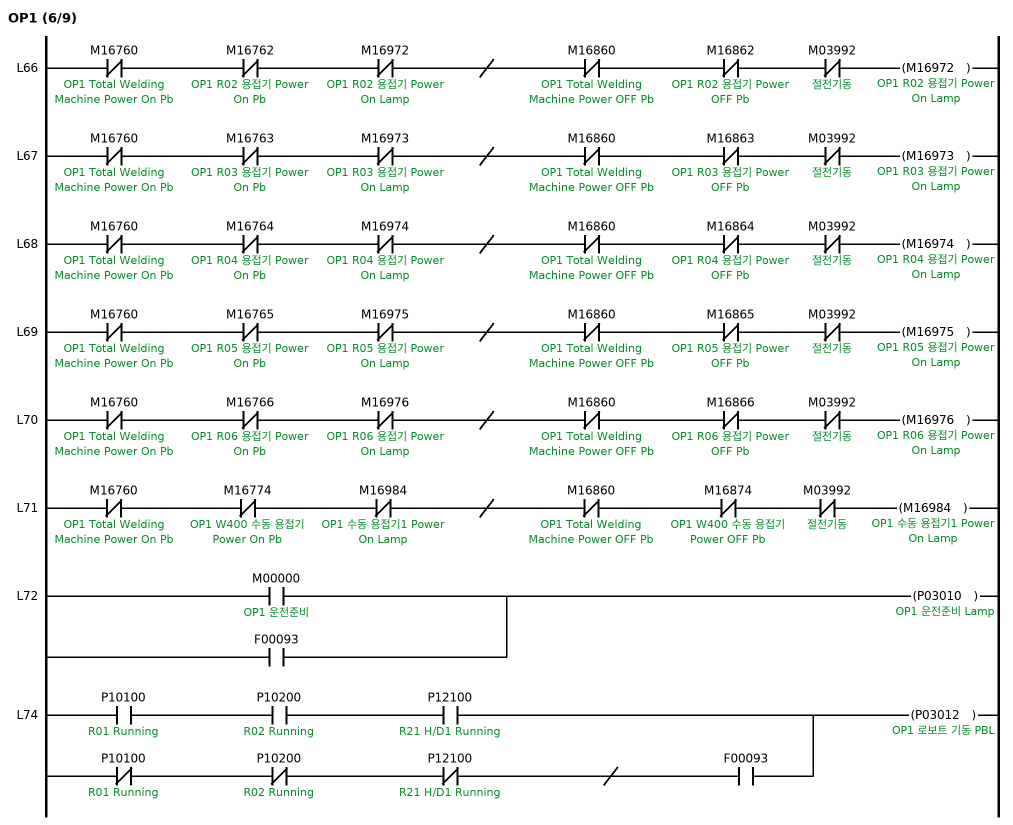
; L66
LOAD NOT  M16760	// OP1 Total Welding Machine Power On Pb
AND NOT   M16762	// OP1 R02 용접기 Power On Pb
AND NOT   M16972	// OP1 R02 용접기 Power On Lamp
NOT
AND NOT   M16860	// OP1 Total Welding Machine Power OFF Pb
AND NOT   M16862	// OP1 R02 용접기 Power OFF Pb
AND NOT   M03992	// 절전기동
OUT       M16972	// OP1 R02 용접기 Power On Lamp
; L67
LOAD NOT  M16760	// OP1 Total Welding Machine Power On Pb
AND NOT   M16763	// OP1 R03 용접기 Power On Pb
AND NOT   M16973	// OP1 R03 용접기 Power On Lamp
NOT
AND NOT   M16860	// OP1 Total Welding Machine Power OFF Pb
AND NOT   M16863	// OP1 R03 용접기 Power OFF Pb
AND NOT   M03992	// 절전기동
OUT       M16973	// OP1 R03 용접기 Power On Lamp
; L68
LOAD NOT  M16760	// OP1 Total Welding Machine Power On Pb
AND NOT   M16764	// OP1 R04 용접기 Power On Pb
AND NOT   M16974	// OP1 R04 용접기 Power On Lamp
NOT
AND NOT   M16860	// OP1 Total Welding Machine Power OFF Pb
AND NOT   M16864	// OP1 R04 용접기 Power OFF Pb
AND NOT   M03992	// 절전기동
OUT       M16974	// OP1 R04 용접기 Power On Lamp
; L69
LOAD NOT  M16760	// OP1 Total Welding Machine Power On Pb
AND NOT   M16765	// OP1 R05 용접기 Power On Pb
AND NOT   M16975	// OP1 R05 용접기 Power On Lamp
NOT
AND NOT   M16860	// OP1 Total Welding Machine Power OFF Pb
AND NOT   M16865	// OP1 R05 용접기 Power OFF Pb
AND NOT   M03992	// 절전기동
OUT       M16975	// OP1 R05 용접기 Power On Lamp
; L70
LOAD NOT  M16760	// OP1 Total Welding Machine Power On Pb
AND NOT   M16766	// OP1 R06 용접기 Power On Pb
AND NOT   M16976	// OP1 R06 용접기 Power On Lamp
NOT
AND NOT   M16860	// OP1 Total Welding Machine Power OFF Pb
AND NOT   M16866	// OP1 R06 용접기 Power OFF Pb
AND NOT   M03992	// 절전기동
OUT       M16976	// OP1 R06 용접기 Power On Lamp
; L71
LOAD NOT  M16760	// OP1 Total Welding Machine Power On Pb
AND NOT   M16774	// OP1 W400 수동 용접기 Power On Pb
AND NOT   M16984	// OP1 수동 용접기1 Power On Lamp
NOT
AND NOT   M16860	// OP1 Total Welding Machine Power OFF Pb
AND NOT   M16874	// OP1 W400 수동 용접기 Power OFF Pb
AND NOT   M03992	// 절전기동
OUT       M16984	// OP1 수동 용접기1 Power On Lamp
; L72
LOAD      M00000	// OP1 운전준비
OR        F00093
OUT       P03010	// OP1 운전준비 Lamp
; L74
LOAD      P10100	// R01 Running
AND       P10200	// R02 Running
AND       P12100	// R21 H/D1 Running
LOAD NOT  P10100	// R01 Running
AND NOT   P10200	// R02 Running
AND NOT   P12100	// R21 H/D1 Running
NOT
AND       F00093
OR LOAD
OUT       P03012	// OP1 로보트 기동 PBL

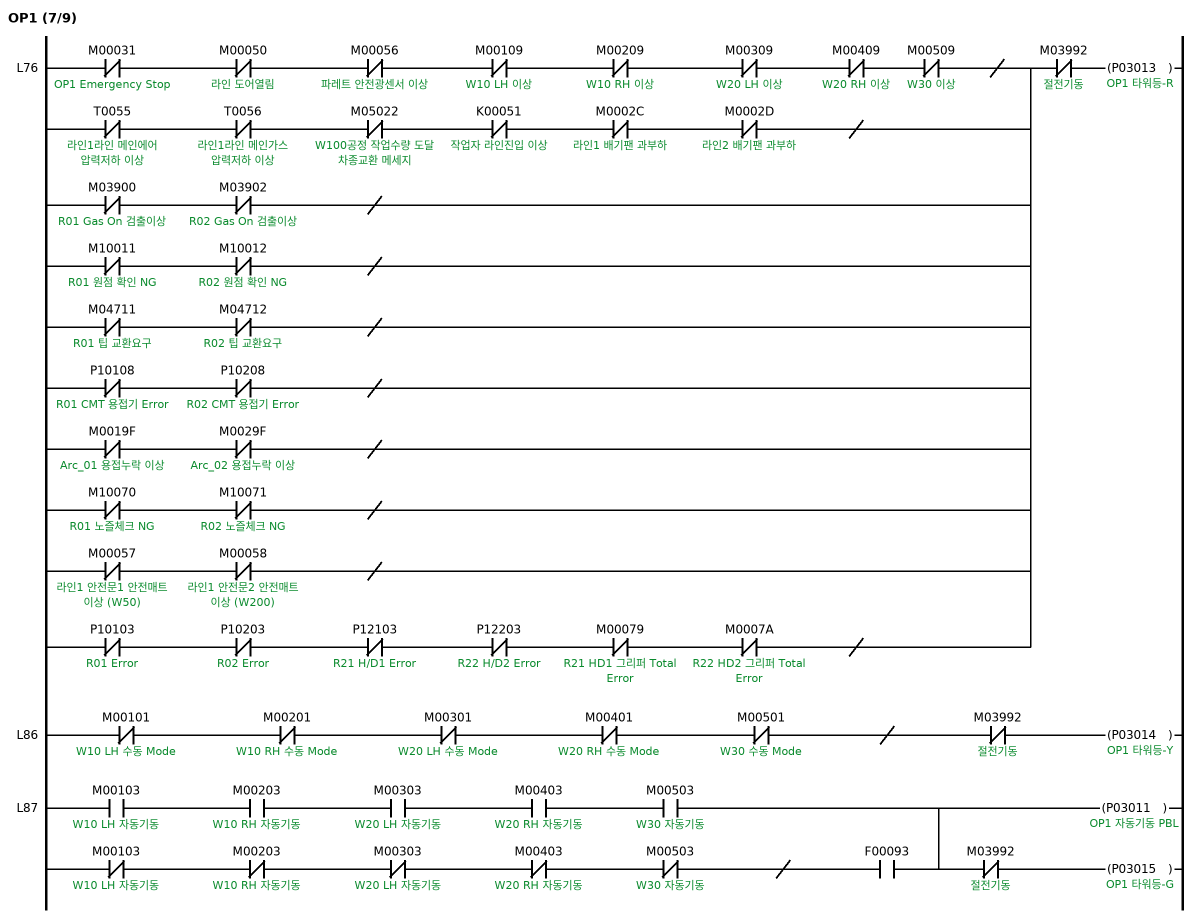
; L76
LOAD NOT  M00031	// OP1 Emergency Stop
AND NOT   M00050	// 라인 도어열림
AND NOT   M00056	// 파레트 안전광센서 이상
AND NOT   M00109	// W10 LH 이상
AND NOT   M00209	// W10 RH 이상
AND NOT   M00309	// W20 LH 이상
AND NOT   M00409	// W20 RH 이상
AND NOT   M00509	// W30 이상
NOT
LOAD NOT  T0055	// 라인1라인 메인에어 압력저하 이상
AND NOT   T0056	// 라인1라인 메인가스 압력저하 이상
AND NOT   M05022	// W100공정 작업수량 도달 차종교환 메세지
AND NOT   K00051	//  작업자 라인진입 이상
AND NOT   M0002C	// 라인1 배기팬 과부하
AND NOT   M0002D	// 라인2 배기팬 과부하
NOT
OR LOAD
LOAD NOT  M03900	// R01 Gas On 검출이상
AND NOT   M03902	// R02 Gas On 검출이상
NOT
OR LOAD
LOAD NOT  M10011	// R01 원점 확인 NG
AND NOT   M10012	// R02 원점 확인 NG
NOT
OR LOAD
LOAD NOT  M04711	// R01 팁 교환요구
AND NOT   M04712	// R02 팁 교환요구
NOT
OR LOAD
LOAD NOT  P10108	// R01 CMT 용접기 Error
AND NOT   P10208	// R02 CMT 용접기 Error
NOT
OR LOAD
LOAD NOT  M0019F	// Arc_01 용접누락 이상
AND NOT   M0029F	// Arc_02 용접누락 이상
NOT
OR LOAD
LOAD NOT  M10070	// R01 노즐체크 NG
AND NOT   M10071	// R02 노즐체크 NG
NOT
OR LOAD
LOAD NOT  M00057	// 라인1 안전문1 안전매트 이상 (W50)
AND NOT   M00058	// 라인1 안전문2 안전매트 이상 (W200)
NOT
OR LOAD
LOAD NOT  P10103	// R01 Error
AND NOT   P10203	// R02 Error
AND NOT   P12103	// R21 H/D1 Error
AND NOT   P12203	// R22 H/D2 Error
AND NOT   M00079	// R21 HD1 그리퍼 Total Error 
AND NOT   M0007A	// R22 HD2 그리퍼 Total Error 
NOT
OR LOAD
AND NOT   M03992	// 절전기동
OUT       P03013	// OP1 타워등-R
; L86
LOAD NOT  M00101	// W10 LH 수동 Mode
AND NOT   M00201	// W10 RH 수동 Mode
AND NOT   M00301	// W20 LH 수동 Mode
AND NOT   M00401	// W20 RH 수동 Mode
AND NOT   M00501	// W30 수동 Mode
NOT
AND NOT   M03992	// 절전기동
OUT       P03014	// OP1 타워등-Y
; L87
LOAD      M00103	// W10 LH 자동기동
AND       M00203	// W10 RH 자동기동
AND       M00303	// W20 LH 자동기동
AND       M00403	// W20 RH 자동기동
AND       M00503	// W30 자동기동
LOAD NOT  M00103	// W10 LH 자동기동
AND NOT   M00203	// W10 RH 자동기동
AND NOT   M00303	// W20 LH 자동기동
AND NOT   M00403	// W20 RH 자동기동
AND NOT   M00503	// W30 자동기동
NOT
AND       F00093
OR LOAD
OUT       P03011	// OP1 자동기동 PBL
AND NOT   M03992	// 절전기동
OUT       P03015	// OP1 타워등-G

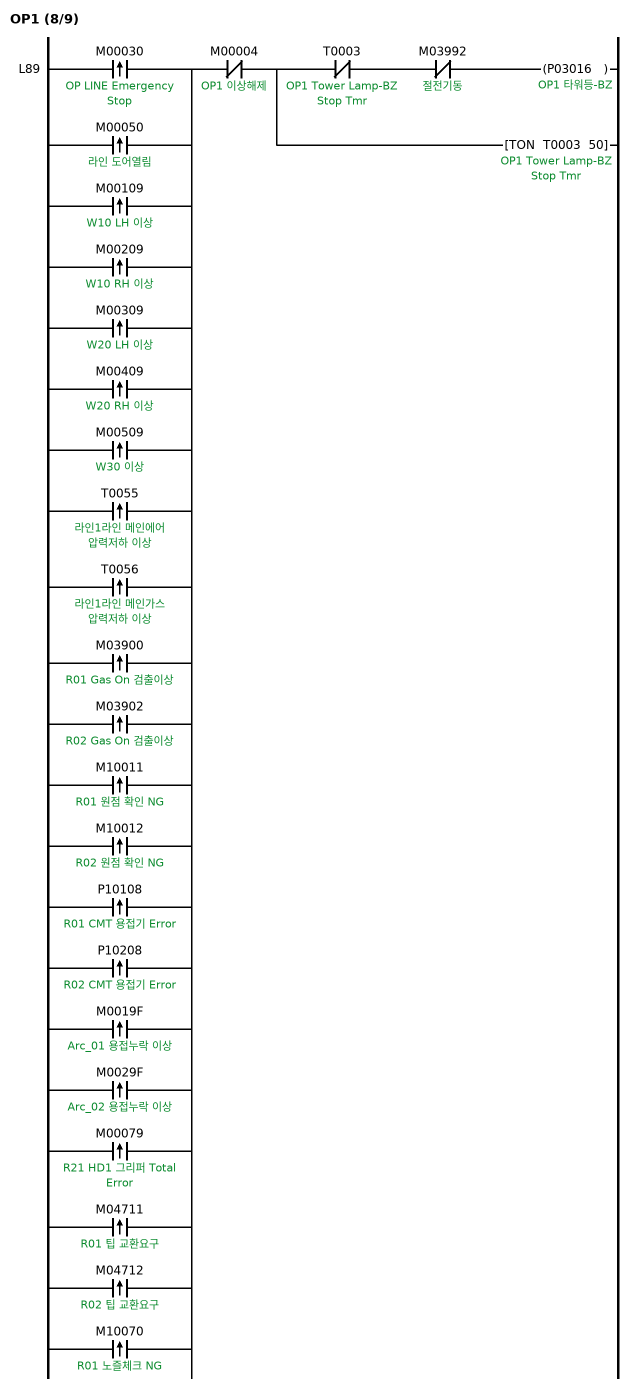

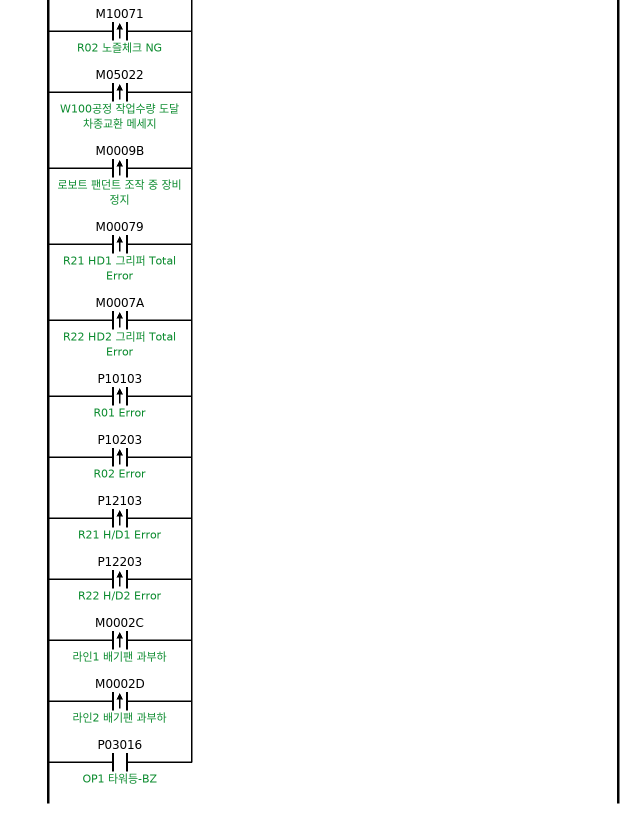
; L89
LOADP     M00030	// OP LINE Emergency Stop
ORP       M00050	// 라인 도어열림
ORP       M00109	// W10 LH 이상
ORP       M00209	// W10 RH 이상
ORP       M00309	// W20 LH 이상
ORP       M00409	// W20 RH 이상
ORP       M00509	// W30 이상
ORP       T0055	// 라인1라인 메인에어 압력저하 이상
ORP       T0056	// 라인1라인 메인가스 압력저하 이상
ORP       M03900	// R01 Gas On 검출이상
ORP       M03902	// R02 Gas On 검출이상
ORP       M10011	// R01 원점 확인 NG
ORP       M10012	// R02 원점 확인 NG
ORP       P10108	// R01 CMT 용접기 Error
ORP       P10208	// R02 CMT 용접기 Error
ORP       M0019F	// Arc_01 용접누락 이상
ORP       M0029F	// Arc_02 용접누락 이상
ORP       M00079	// R21 HD1 그리퍼 Total Error 
ORP       M04711	// R01 팁 교환요구
ORP       M04712	// R02 팁 교환요구
ORP       M10070	// R01 노즐체크 NG
ORP       M10071	// R02 노즐체크 NG
ORP       M05022	// W100공정 작업수량 도달 차종교환 메세지
ORP       M0009B	// 로보트 팬던트 조작 중 장비 정지
ORP       M00079	// R21 HD1 그리퍼 Total Error 
ORP       M0007A	// R22 HD2 그리퍼 Total Error 
ORP       P10103	// R01 Error
ORP       P10203	// R02 Error
ORP       P12103	// R21 H/D1 Error
ORP       P12203	// R22 H/D2 Error
ORP       M0002C	// 라인1 배기팬 과부하
ORP       M0002D	// 라인2 배기팬 과부하
OR        P03016	// OP1 타워등-BZ
AND NOT   M00004	// OP1 이상해제
MPUSH
AND NOT   T0003	// OP1 Tower Lamp-BZ Stop Tmr
AND NOT   M03992	// 절전기동
OUT       P03016	// OP1 타워등-BZ
MPOP
TON       T0003 50	// OP1 Tower Lamp-BZ Stop Tmr

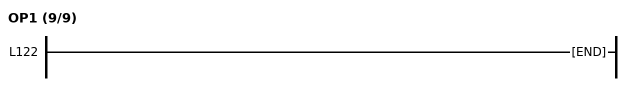
; L122
END

PROGRAM OP2 (task: 스캔 프로그램)

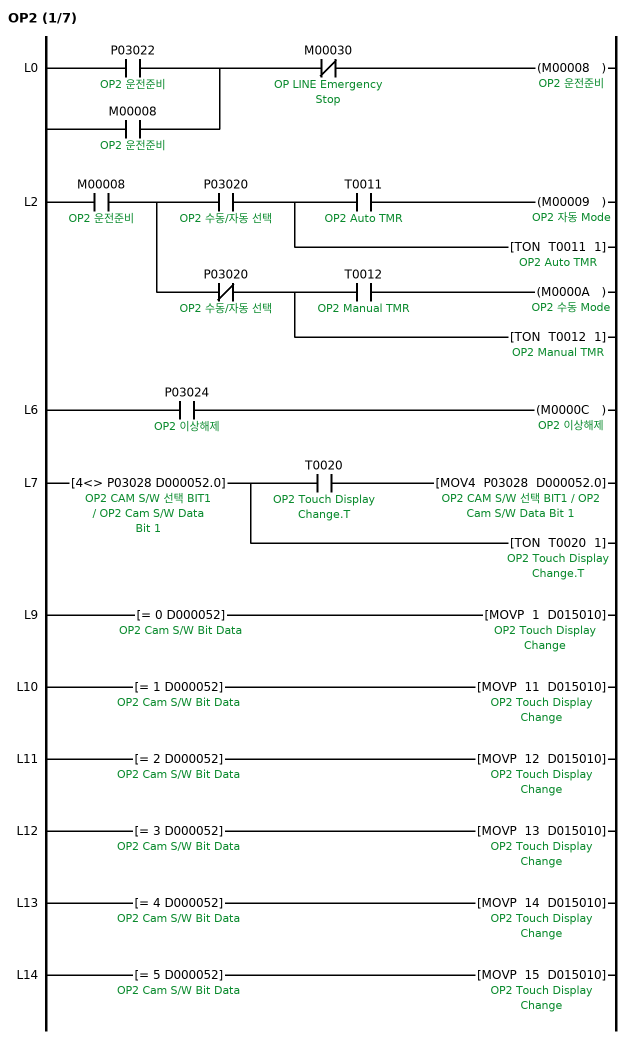
; L0
LOAD      P03022	// OP2 운전준비
OR        M00008	// OP2 운전준비
AND NOT   M00030	// OP LINE Emergency Stop
OUT       M00008	// OP2 운전준비
; L2
LOAD      M00008	// OP2 운전준비
MPUSH
AND       P03020	// OP2 수동/자동 선택
MPUSH
AND       T0011	// OP2 Auto TMR
OUT       M00009	// OP2 자동 Mode
MPOP
TON       T0011 1	// OP2 Auto TMR
MPOP
AND NOT   P03020	// OP2 수동/자동 선택
MPUSH
AND       T0012	// OP2 Manual TMR
OUT       M0000A	// OP2 수동 Mode
MPOP
TON       T0012 1	// OP2 Manual TMR
; L6
LOAD      P03024	// OP2 이상해제
OUT       M0000C	// OP2 이상해제
; L7
LOAD4<>   P03028 D000052.0	// OP2 CAM S/W 선택 BIT1 / OP2 Cam S/W Data Bit 1
MPUSH
AND       T0020	// OP2 Touch Display Change.T
MOV4      P03028 D000052.0	// OP2 CAM S/W 선택 BIT1 / OP2 Cam S/W Data Bit 1
MPOP
TON       T0020 1	// OP2 Touch Display Change.T
; L9
LOAD=     0 D000052	// OP2 Cam S/W Bit Data
MOVP      1 D015010	// OP2 Touch Display Change
; L10
LOAD=     1 D000052	// OP2 Cam S/W Bit Data
MOVP      11 D015010	// OP2 Touch Display Change
; L11
LOAD=     2 D000052	// OP2 Cam S/W Bit Data
MOVP      12 D015010	// OP2 Touch Display Change
; L12
LOAD=     3 D000052	// OP2 Cam S/W Bit Data
MOVP      13 D015010	// OP2 Touch Display Change
; L13
LOAD=     4 D000052	// OP2 Cam S/W Bit Data
MOVP      14 D015010	// OP2 Touch Display Change
; L14
LOAD=     5 D000052	// OP2 Cam S/W Bit Data
MOVP      15 D015010	// OP2 Touch Display Change

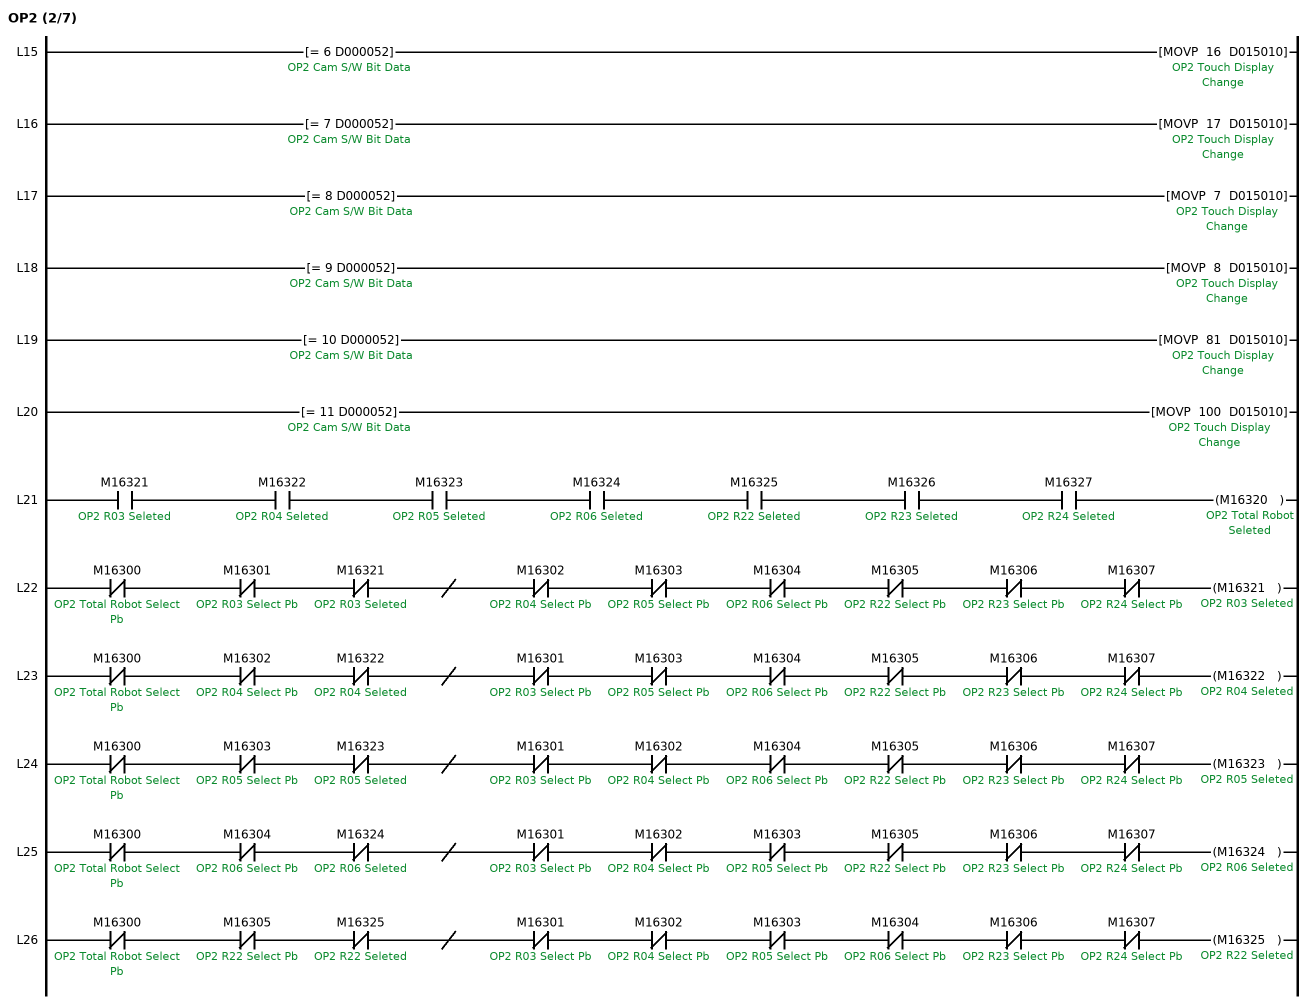
; L15
LOAD=     6 D000052	// OP2 Cam S/W Bit Data
MOVP      16 D015010	// OP2 Touch Display Change
; L16
LOAD=     7 D000052	// OP2 Cam S/W Bit Data
MOVP      17 D015010	// OP2 Touch Display Change
; L17
LOAD=     8 D000052	// OP2 Cam S/W Bit Data
MOVP      7 D015010	// OP2 Touch Display Change
; L18
LOAD=     9 D000052	// OP2 Cam S/W Bit Data
MOVP      8 D015010	// OP2 Touch Display Change
; L19
LOAD=     10 D000052	// OP2 Cam S/W Bit Data
MOVP      81 D015010	// OP2 Touch Display Change
; L20
LOAD=     11 D000052	// OP2 Cam S/W Bit Data
MOVP      100 D015010	// OP2 Touch Display Change
; L21
LOAD      M16321	// OP2 R03 Seleted
AND       M16322	// OP2 R04 Seleted
AND       M16323	// OP2 R05 Seleted
AND       M16324	// OP2 R06 Seleted
AND       M16325	// OP2 R22 Seleted
AND       M16326	// OP2 R23 Seleted
AND       M16327	// OP2 R24 Seleted
OUT       M16320	// OP2 Total Robot Seleted
; L22
LOAD NOT  M16300	// OP2 Total Robot Select Pb
AND NOT   M16301	// OP2 R03 Select Pb
AND NOT   M16321	// OP2 R03 Seleted
NOT
AND NOT   M16302	// OP2 R04 Select Pb
AND NOT   M16303	// OP2 R05 Select Pb
AND NOT   M16304	// OP2 R06 Select Pb
AND NOT   M16305	// OP2 R22 Select Pb
AND NOT   M16306	// OP2 R23 Select Pb
AND NOT   M16307	// OP2 R24 Select Pb
OUT       M16321	// OP2 R03 Seleted
; L23
LOAD NOT  M16300	// OP2 Total Robot Select Pb
AND NOT   M16302	// OP2 R04 Select Pb
AND NOT   M16322	// OP2 R04 Seleted
NOT
AND NOT   M16301	// OP2 R03 Select Pb
AND NOT   M16303	// OP2 R05 Select Pb
AND NOT   M16304	// OP2 R06 Select Pb
AND NOT   M16305	// OP2 R22 Select Pb
AND NOT   M16306	// OP2 R23 Select Pb
AND NOT   M16307	// OP2 R24 Select Pb
OUT       M16322	// OP2 R04 Seleted
; L24
LOAD NOT  M16300	// OP2 Total Robot Select Pb
AND NOT   M16303	// OP2 R05 Select Pb
AND NOT   M16323	// OP2 R05 Seleted
NOT
AND NOT   M16301	// OP2 R03 Select Pb
AND NOT   M16302	// OP2 R04 Select Pb
AND NOT   M16304	// OP2 R06 Select Pb
AND NOT   M16305	// OP2 R22 Select Pb
AND NOT   M16306	// OP2 R23 Select Pb
AND NOT   M16307	// OP2 R24 Select Pb
OUT       M16323	// OP2 R05 Seleted
; L25
LOAD NOT  M16300	// OP2 Total Robot Select Pb
AND NOT   M16304	// OP2 R06 Select Pb
AND NOT   M16324	// OP2 R06 Seleted
NOT
AND NOT   M16301	// OP2 R03 Select Pb
AND NOT   M16302	// OP2 R04 Select Pb
AND NOT   M16303	// OP2 R05 Select Pb
AND NOT   M16305	// OP2 R22 Select Pb
AND NOT   M16306	// OP2 R23 Select Pb
AND NOT   M16307	// OP2 R24 Select Pb
OUT       M16324	// OP2 R06 Seleted
; L26
LOAD NOT  M16300	// OP2 Total Robot Select Pb
AND NOT   M16305	// OP2 R22 Select Pb
AND NOT   M16325	// OP2 R22 Seleted
NOT
AND NOT   M16301	// OP2 R03 Select Pb
AND NOT   M16302	// OP2 R04 Select Pb
AND NOT   M16303	// OP2 R05 Select Pb
AND NOT   M16304	// OP2 R06 Select Pb
AND NOT   M16306	// OP2 R23 Select Pb
AND NOT   M16307	// OP2 R24 Select Pb
OUT       M16325	// OP2 R22 Seleted

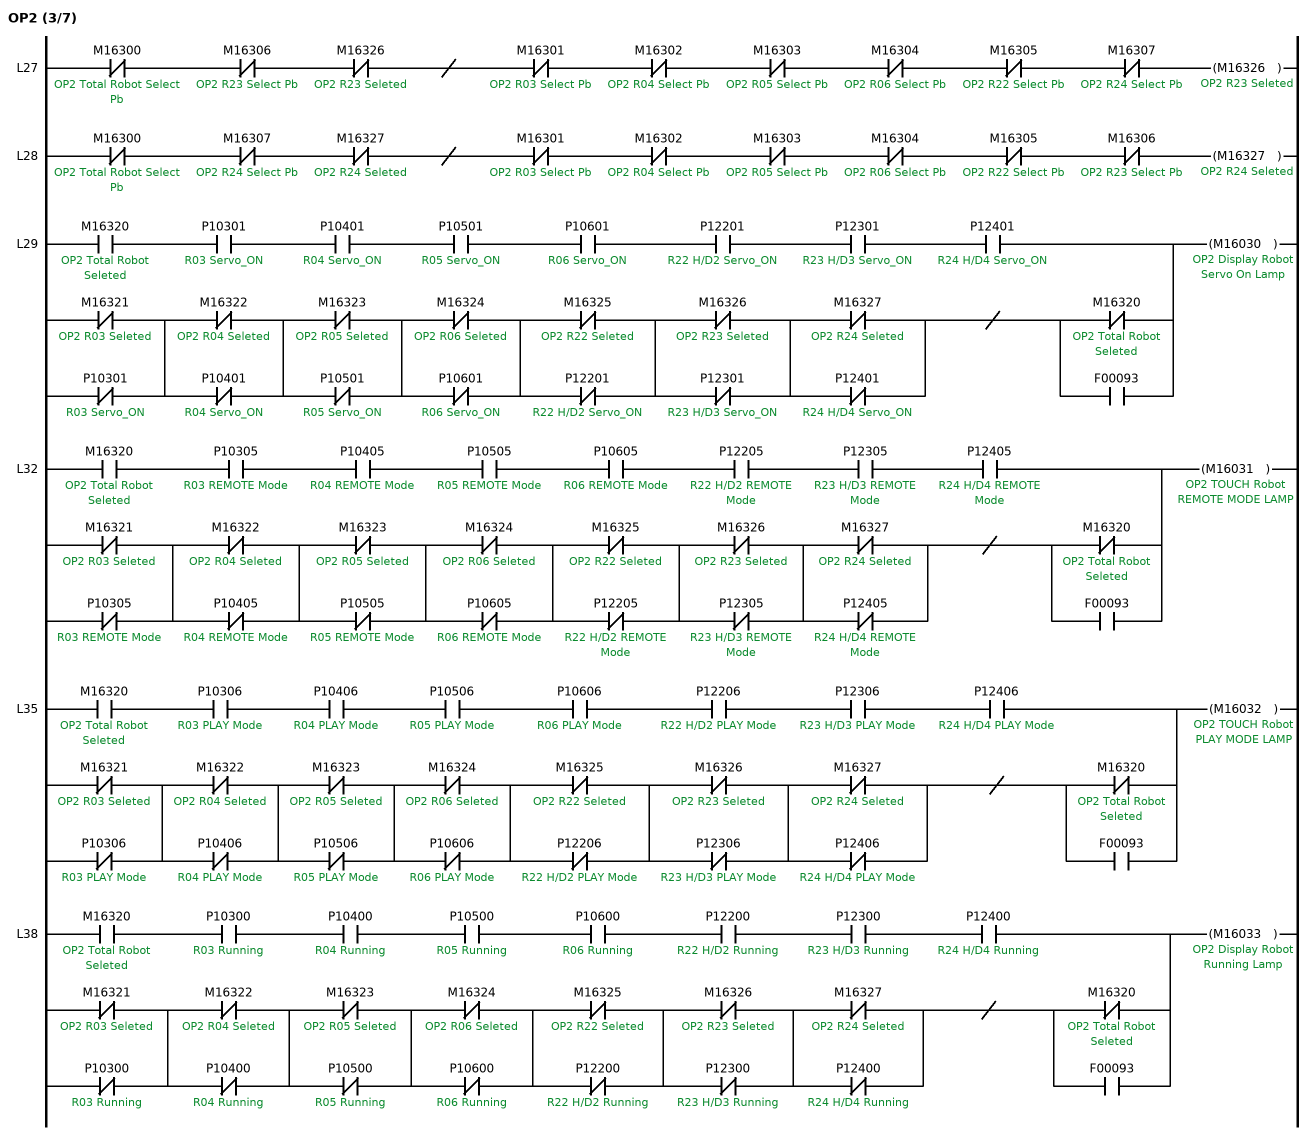
; L27
LOAD NOT  M16300	// OP2 Total Robot Select Pb
AND NOT   M16306	// OP2 R23 Select Pb
AND NOT   M16326	// OP2 R23 Seleted
NOT
AND NOT   M16301	// OP2 R03 Select Pb
AND NOT   M16302	// OP2 R04 Select Pb
AND NOT   M16303	// OP2 R05 Select Pb
AND NOT   M16304	// OP2 R06 Select Pb
AND NOT   M16305	// OP2 R22 Select Pb
AND NOT   M16307	// OP2 R24 Select Pb
OUT       M16326	// OP2 R23 Seleted
; L28
LOAD NOT  M16300	// OP2 Total Robot Select Pb
AND NOT   M16307	// OP2 R24 Select Pb
AND NOT   M16327	// OP2 R24 Seleted
NOT
AND NOT   M16301	// OP2 R03 Select Pb
AND NOT   M16302	// OP2 R04 Select Pb
AND NOT   M16303	// OP2 R05 Select Pb
AND NOT   M16304	// OP2 R06 Select Pb
AND NOT   M16305	// OP2 R22 Select Pb
AND NOT   M16306	// OP2 R23 Select Pb
OUT       M16327	// OP2 R24 Seleted
; L29
LOAD      M16320	// OP2 Total Robot Seleted
AND       P10301	// R03 Servo_ON
AND       P10401	// R04 Servo_ON
AND       P10501	// R05 Servo_ON
AND       P10601	// R06 Servo_ON
AND       P12201	// R22 H/D2 Servo_ON
AND       P12301	// R23 H/D3 Servo_ON
AND       P12401	// R24 H/D4 Servo_ON
LOAD NOT  M16321	// OP2 R03 Seleted
OR NOT    P10301	// R03 Servo_ON
LOAD NOT  M16322	// OP2 R04 Seleted
OR NOT    P10401	// R04 Servo_ON
AND LOAD
LOAD NOT  M16323	// OP2 R05 Seleted
OR NOT    P10501	// R05 Servo_ON
AND LOAD
LOAD NOT  M16324	// OP2 R06 Seleted
OR NOT    P10601	// R06 Servo_ON
AND LOAD
LOAD NOT  M16325	// OP2 R22 Seleted
OR NOT    P12201	// R22 H/D2 Servo_ON
AND LOAD
LOAD NOT  M16326	// OP2 R23 Seleted
OR NOT    P12301	// R23 H/D3 Servo_ON
AND LOAD
LOAD NOT  M16327	// OP2 R24 Seleted
OR NOT    P12401	// R24 H/D4 Servo_ON
AND LOAD
NOT
LOAD NOT  M16320	// OP2 Total Robot Seleted
OR        F00093
AND LOAD
OR LOAD
OUT       M16030	// OP2 Display Robot Servo On Lamp
; L32
LOAD      M16320	// OP2 Total Robot Seleted
AND       P10305	// R03 REMOTE Mode
AND       P10405	// R04 REMOTE Mode
AND       P10505	// R05 REMOTE Mode
AND       P10605	// R06 REMOTE Mode
AND       P12205	// R22 H/D2 REMOTE Mode
AND       P12305	// R23 H/D3 REMOTE Mode
AND       P12405	// R24 H/D4 REMOTE Mode
LOAD NOT  M16321	// OP2 R03 Seleted
OR NOT    P10305	// R03 REMOTE Mode
LOAD NOT  M16322	// OP2 R04 Seleted
OR NOT    P10405	// R04 REMOTE Mode
AND LOAD
LOAD NOT  M16323	// OP2 R05 Seleted
OR NOT    P10505	// R05 REMOTE Mode
AND LOAD
LOAD NOT  M16324	// OP2 R06 Seleted
OR NOT    P10605	// R06 REMOTE Mode
AND LOAD
LOAD NOT  M16325	// OP2 R22 Seleted
OR NOT    P12205	// R22 H/D2 REMOTE Mode
AND LOAD
LOAD NOT  M16326	// OP2 R23 Seleted
OR NOT    P12305	// R23 H/D3 REMOTE Mode
AND LOAD
LOAD NOT  M16327	// OP2 R24 Seleted
OR NOT    P12405	// R24 H/D4 REMOTE Mode
AND LOAD
NOT
LOAD NOT  M16320	// OP2 Total Robot Seleted
OR        F00093
AND LOAD
OR LOAD
OUT       M16031	// OP2 TOUCH Robot REMOTE MODE LAMP
; L35
LOAD      M16320	// OP2 Total Robot Seleted
AND       P10306	// R03 PLAY Mode
AND       P10406	// R04 PLAY Mode
AND       P10506	// R05 PLAY Mode
AND       P10606	// R06 PLAY Mode
AND       P12206	// R22 H/D2 PLAY Mode
AND       P12306	// R23 H/D3 PLAY Mode
AND       P12406	// R24 H/D4 PLAY Mode
LOAD NOT  M16321	// OP2 R03 Seleted
OR NOT    P10306	// R03 PLAY Mode
LOAD NOT  M16322	// OP2 R04 Seleted
OR NOT    P10406	// R04 PLAY Mode
AND LOAD
LOAD NOT  M16323	// OP2 R05 Seleted
OR NOT    P10506	// R05 PLAY Mode
AND LOAD
LOAD NOT  M16324	// OP2 R06 Seleted
OR NOT    P10606	// R06 PLAY Mode
AND LOAD
LOAD NOT  M16325	// OP2 R22 Seleted
OR NOT    P12206	// R22 H/D2 PLAY Mode
AND LOAD
LOAD NOT  M16326	// OP2 R23 Seleted
OR NOT    P12306	// R23 H/D3 PLAY Mode
AND LOAD
LOAD NOT  M16327	// OP2 R24 Seleted
OR NOT    P12406	// R24 H/D4 PLAY Mode
AND LOAD
NOT
LOAD NOT  M16320	// OP2 Total Robot Seleted
OR        F00093
AND LOAD
OR LOAD
OUT       M16032	// OP2 TOUCH Robot PLAY MODE LAMP
; L38
LOAD      M16320	// OP2 Total Robot Seleted
AND       P10300	// R03 Running
AND       P10400	// R04 Running
AND       P10500	// R05 Running
AND       P10600	// R06 Running
AND       P12200	// R22 H/D2 Running
AND       P12300	// R23 H/D3 Running
AND       P12400	// R24 H/D4 Running
LOAD NOT  M16321	// OP2 R03 Seleted
OR NOT    P10300	// R03 Running
LOAD NOT  M16322	// OP2 R04 Seleted
OR NOT    P10400	// R04 Running
AND LOAD
LOAD NOT  M16323	// OP2 R05 Seleted
OR NOT    P10500	// R05 Running
AND LOAD
LOAD NOT  M16324	// OP2 R06 Seleted
OR NOT    P10600	// R06 Running
AND LOAD
LOAD NOT  M16325	// OP2 R22 Seleted
OR NOT    P12200	// R22 H/D2 Running
AND LOAD
LOAD NOT  M16326	// OP2 R23 Seleted
OR NOT    P12300	// R23 H/D3 Running
AND LOAD
LOAD NOT  M16327	// OP2 R24 Seleted
OR NOT    P12400	// R24 H/D4 Running
AND LOAD
NOT
LOAD NOT  M16320	// OP2 Total Robot Seleted
OR        F00093
AND LOAD
OR LOAD
OUT       M16033	// OP2 Display Robot Running Lamp

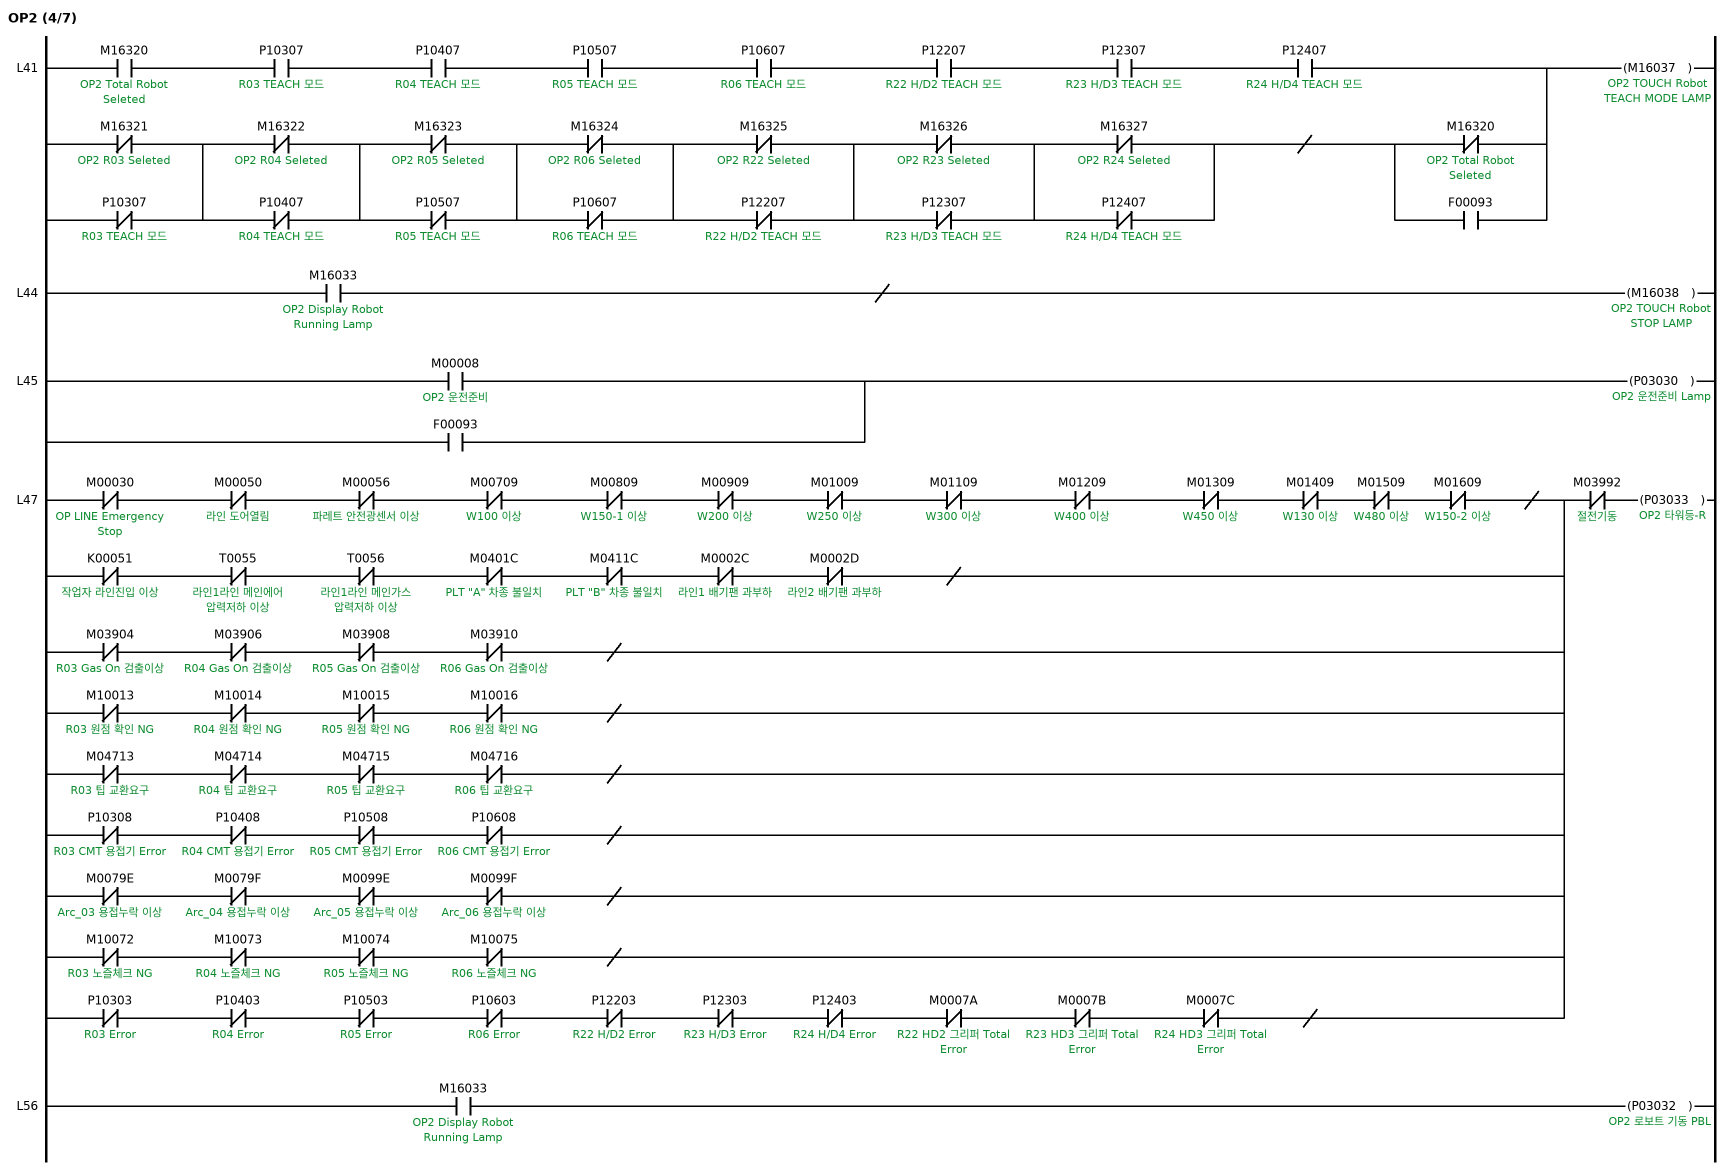
; L41
LOAD      M16320	// OP2 Total Robot Seleted
AND       P10307	// R03 TEACH 모드
AND       P10407	// R04 TEACH 모드
AND       P10507	// R05 TEACH 모드
AND       P10607	// R06 TEACH 모드
AND       P12207	// R22 H/D2 TEACH 모드
AND       P12307	// R23 H/D3 TEACH 모드
AND       P12407	// R24 H/D4 TEACH 모드
LOAD NOT  M16321	// OP2 R03 Seleted
OR NOT    P10307	// R03 TEACH 모드
LOAD NOT  M16322	// OP2 R04 Seleted
OR NOT    P10407	// R04 TEACH 모드
AND LOAD
LOAD NOT  M16323	// OP2 R05 Seleted
OR NOT    P10507	// R05 TEACH 모드
AND LOAD
LOAD NOT  M16324	// OP2 R06 Seleted
OR NOT    P10607	// R06 TEACH 모드
AND LOAD
LOAD NOT  M16325	// OP2 R22 Seleted
OR NOT    P12207	// R22 H/D2 TEACH 모드
AND LOAD
LOAD NOT  M16326	// OP2 R23 Seleted
OR NOT    P12307	// R23 H/D3 TEACH 모드
AND LOAD
LOAD NOT  M16327	// OP2 R24 Seleted
OR NOT    P12407	// R24 H/D4 TEACH 모드
AND LOAD
NOT
LOAD NOT  M16320	// OP2 Total Robot Seleted
OR        F00093
AND LOAD
OR LOAD
OUT       M16037	// OP2 TOUCH Robot TEACH MODE LAMP
; L44
LOAD      M16033	// OP2 Display Robot Running Lamp
NOT
OUT       M16038	// OP2 TOUCH Robot STOP LAMP
; L45
LOAD      M00008	// OP2 운전준비
OR        F00093
OUT       P03030	// OP2 운전준비 Lamp
; L47
LOAD NOT  M00030	// OP LINE Emergency Stop
AND NOT   M00050	// 라인 도어열림
AND NOT   M00056	// 파레트 안전광센서 이상
AND NOT   M00709	// W100 이상
AND NOT   M00809	// W150-1 이상
AND NOT   M00909	// W200 이상
AND NOT   M01009	// W250 이상
AND NOT   M01109	// W300 이상
AND NOT   M01209	// W400 이상
AND NOT   M01309	// W450 이상
AND NOT   M01409	// W130 이상
AND NOT   M01509	// W480 이상
AND NOT   M01609	// W150-2 이상
NOT
LOAD NOT  K00051	//  작업자 라인진입 이상
AND NOT   T0055	// 라인1라인 메인에어 압력저하 이상
AND NOT   T0056	// 라인1라인 메인가스 압력저하 이상
AND NOT   M0401C	// PLT "A" 차종 불일치
AND NOT   M0411C	// PLT "B" 차종 불일치
AND NOT   M0002C	// 라인1 배기팬 과부하
AND NOT   M0002D	// 라인2 배기팬 과부하
NOT
OR LOAD
LOAD NOT  M03904	// R03 Gas On 검출이상
AND NOT   M03906	// R04 Gas On 검출이상
AND NOT   M03908	// R05 Gas On 검출이상
AND NOT   M03910	// R06 Gas On 검출이상
NOT
OR LOAD
LOAD NOT  M10013	// R03 원점 확인 NG
AND NOT   M10014	// R04 원점 확인 NG
AND NOT   M10015	// R05 원점 확인 NG
AND NOT   M10016	// R06 원점 확인 NG
NOT
OR LOAD
LOAD NOT  M04713	// R03 팁 교환요구
AND NOT   M04714	// R04 팁 교환요구
AND NOT   M04715	// R05 팁 교환요구
AND NOT   M04716	// R06 팁 교환요구
NOT
OR LOAD
LOAD NOT  P10308	// R03 CMT 용접기 Error
AND NOT   P10408	// R04 CMT 용접기 Error
AND NOT   P10508	// R05 CMT 용접기 Error
AND NOT   P10608	// R06 CMT 용접기 Error
NOT
OR LOAD
LOAD NOT  M0079E	// Arc_03 용접누락 이상
AND NOT   M0079F	// Arc_04 용접누락 이상
AND NOT   M0099E	// Arc_05 용접누락 이상
AND NOT   M0099F	// Arc_06 용접누락 이상
NOT
OR LOAD
LOAD NOT  M10072	// R03 노즐체크 NG
AND NOT   M10073	// R04 노즐체크 NG
AND NOT   M10074	// R05 노즐체크 NG
AND NOT   M10075	// R06 노즐체크 NG
NOT
OR LOAD
LOAD NOT  P10303	// R03 Error
AND NOT   P10403	// R04 Error
AND NOT   P10503	// R05 Error
AND NOT   P10603	// R06 Error
AND NOT   P12203	// R22 H/D2 Error
AND NOT   P12303	// R23 H/D3 Error
AND NOT   P12403	// R24 H/D4 Error
AND NOT   M0007A	// R22 HD2 그리퍼 Total Error 
AND NOT   M0007B	// R23 HD3 그리퍼 Total Error 
AND NOT   M0007C	// R24 HD3 그리퍼 Total Error 
NOT
OR LOAD
AND NOT   M03992	// 절전기동
OUT       P03033	// OP2 타워등-R
; L56
LOAD      M16033	// OP2 Display Robot Running Lamp
OUT       P03032	// OP2 로보트 기동 PBL

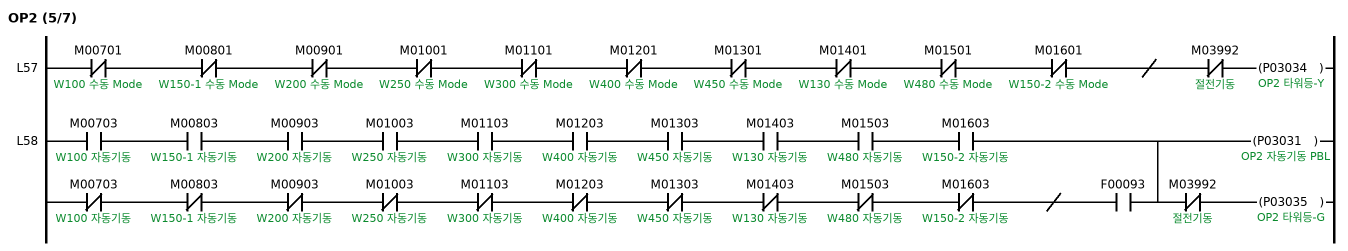
; L57
LOAD NOT  M00701	// W100 수동 Mode
AND NOT   M00801	// W150-1 수동 Mode
AND NOT   M00901	// W200 수동 Mode
AND NOT   M01001	// W250 수동 Mode
AND NOT   M01101	// W300 수동 Mode
AND NOT   M01201	// W400 수동 Mode
AND NOT   M01301	// W450 수동 Mode
AND NOT   M01401	// W130 수동 Mode
AND NOT   M01501	// W480 수동 Mode
AND NOT   M01601	// W150-2 수동 Mode
NOT
AND NOT   M03992	// 절전기동
OUT       P03034	// OP2 타워등-Y
; L58
LOAD      M00703	// W100 자동기동
AND       M00803	// W150-1 자동기동
AND       M00903	// W200 자동기동
AND       M01003	// W250 자동기동
AND       M01103	// W300 자동기동
AND       M01203	// W400 자동기동
AND       M01303	// W450 자동기동
AND       M01403	// W130 자동기동
AND       M01503	// W480 자동기동
AND       M01603	// W150-2 자동기동
LOAD NOT  M00703	// W100 자동기동
AND NOT   M00803	// W150-1 자동기동
AND NOT   M00903	// W200 자동기동
AND NOT   M01003	// W250 자동기동
AND NOT   M01103	// W300 자동기동
AND NOT   M01203	// W400 자동기동
AND NOT   M01303	// W450 자동기동
AND NOT   M01403	// W130 자동기동
AND NOT   M01503	// W480 자동기동
AND NOT   M01603	// W150-2 자동기동
NOT
AND       F00093
OR LOAD
OUT       P03031	// OP2 자동기동 PBL
AND NOT   M03992	// 절전기동
OUT       P03035	// OP2 타워등-G

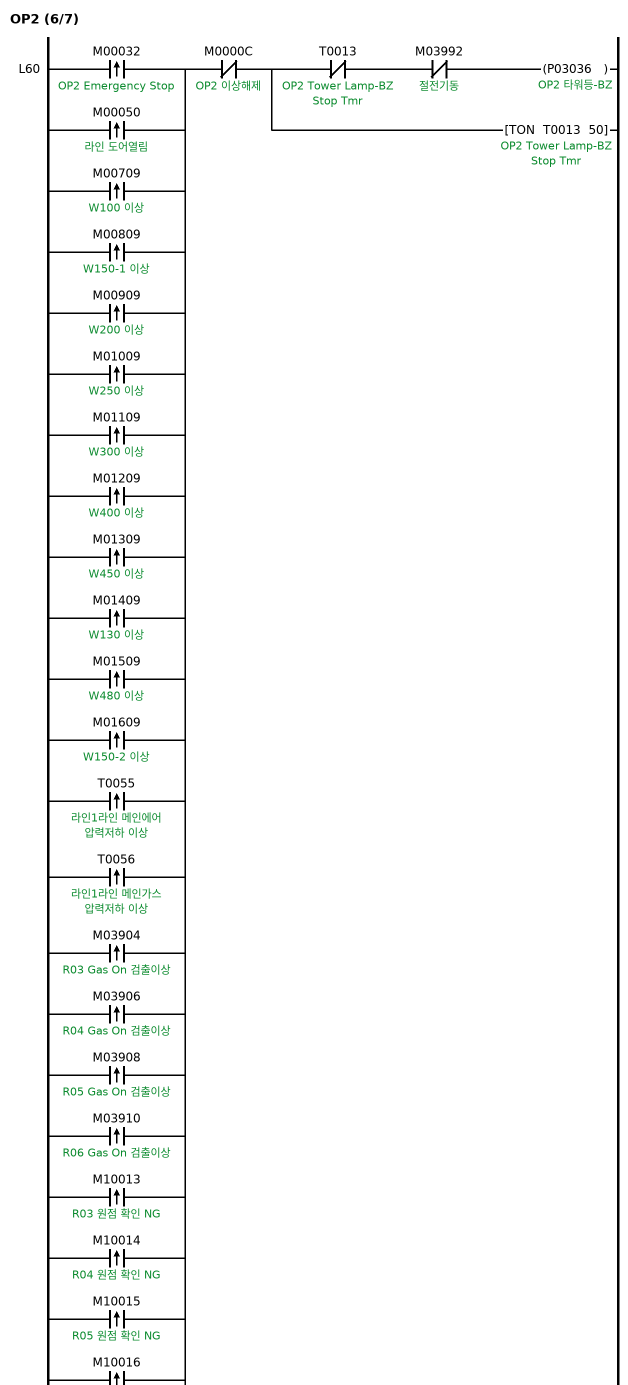

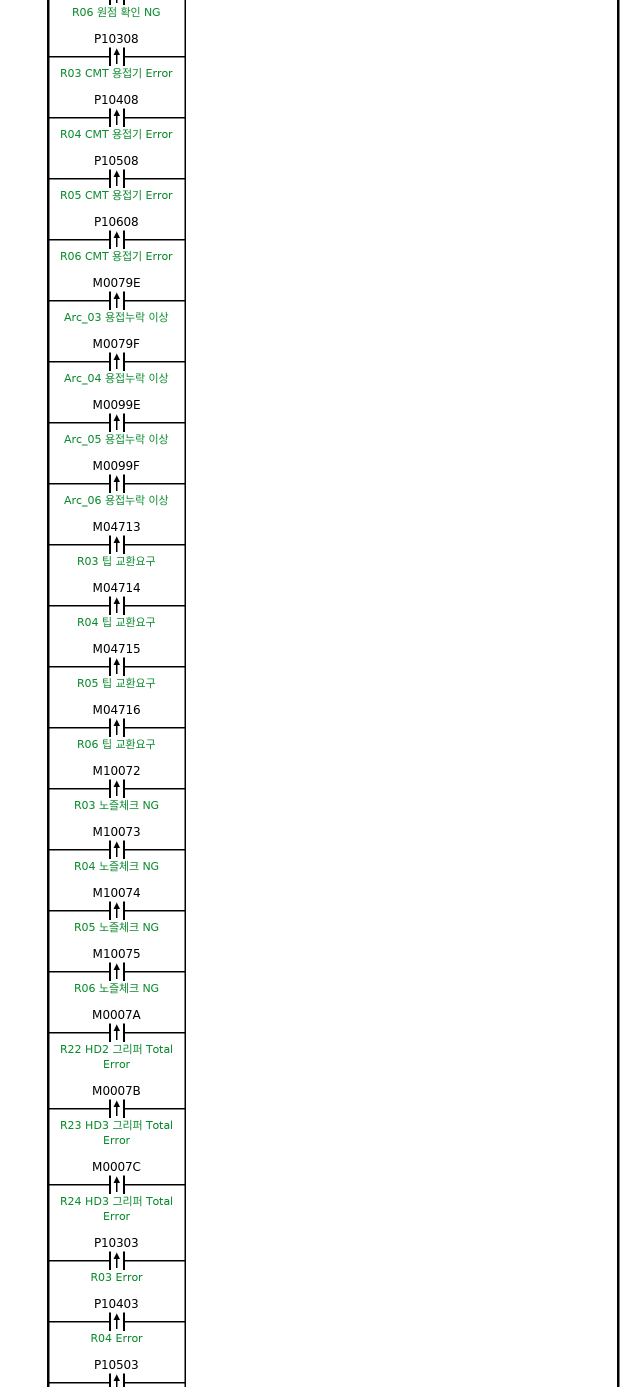

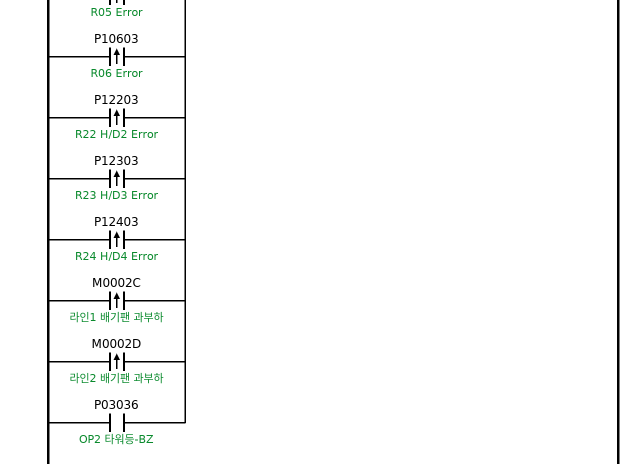
; L60
LOADP     M00032	// OP2 Emergency Stop
ORP       M00050	// 라인 도어열림
ORP       M00709	// W100 이상
ORP       M00809	// W150-1 이상
ORP       M00909	// W200 이상
ORP       M01009	// W250 이상
ORP       M01109	// W300 이상
ORP       M01209	// W400 이상
ORP       M01309	// W450 이상
ORP       M01409	// W130 이상
ORP       M01509	// W480 이상
ORP       M01609	// W150-2 이상
ORP       T0055	// 라인1라인 메인에어 압력저하 이상
ORP       T0056	// 라인1라인 메인가스 압력저하 이상
ORP       M03904	// R03 Gas On 검출이상
ORP       M03906	// R04 Gas On 검출이상
ORP       M03908	// R05 Gas On 검출이상
ORP       M03910	// R06 Gas On 검출이상
ORP       M10013	// R03 원점 확인 NG
ORP       M10014	// R04 원점 확인 NG
ORP       M10015	// R05 원점 확인 NG
ORP       M10016	// R06 원점 확인 NG
ORP       P10308	// R03 CMT 용접기 Error
ORP       P10408	// R04 CMT 용접기 Error
ORP       P10508	// R05 CMT 용접기 Error
ORP       P10608	// R06 CMT 용접기 Error
ORP       M0079E	// Arc_03 용접누락 이상
ORP       M0079F	// Arc_04 용접누락 이상
ORP       M0099E	// Arc_05 용접누락 이상
ORP       M0099F	// Arc_06 용접누락 이상
ORP       M04713	// R03 팁 교환요구
ORP       M04714	// R04 팁 교환요구
ORP       M04715	// R05 팁 교환요구
ORP       M04716	// R06 팁 교환요구
ORP       M10072	// R03 노즐체크 NG
ORP       M10073	// R04 노즐체크 NG
ORP       M10074	// R05 노즐체크 NG
ORP       M10075	// R06 노즐체크 NG
ORP       M0007A	// R22 HD2 그리퍼 Total Error 
ORP       M0007B	// R23 HD3 그리퍼 Total Error 
ORP       M0007C	// R24 HD3 그리퍼 Total Error 
ORP       P10303	// R03 Error
ORP       P10403	// R04 Error
ORP       P10503	// R05 Error
ORP       P10603	// R06 Error
ORP       P12203	// R22 H/D2 Error
ORP       P12303	// R23 H/D3 Error
ORP       P12403	// R24 H/D4 Error
ORP       M0002C	// 라인1 배기팬 과부하
ORP       M0002D	// 라인2 배기팬 과부하
OR        P03036	// OP2 타워등-BZ
AND NOT   M0000C	// OP2 이상해제
MPUSH
AND NOT   T0013	// OP2 Tower Lamp-BZ Stop Tmr
AND NOT   M03992	// 절전기동
OUT       P03036	// OP2 타워등-BZ
MPOP
TON       T0013 50	// OP2 Tower Lamp-BZ Stop Tmr

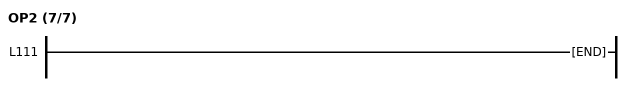
; L111
END

PROGRAM MAIN_STN1_W10_LH(M100) (task: 스캔 프로그램)

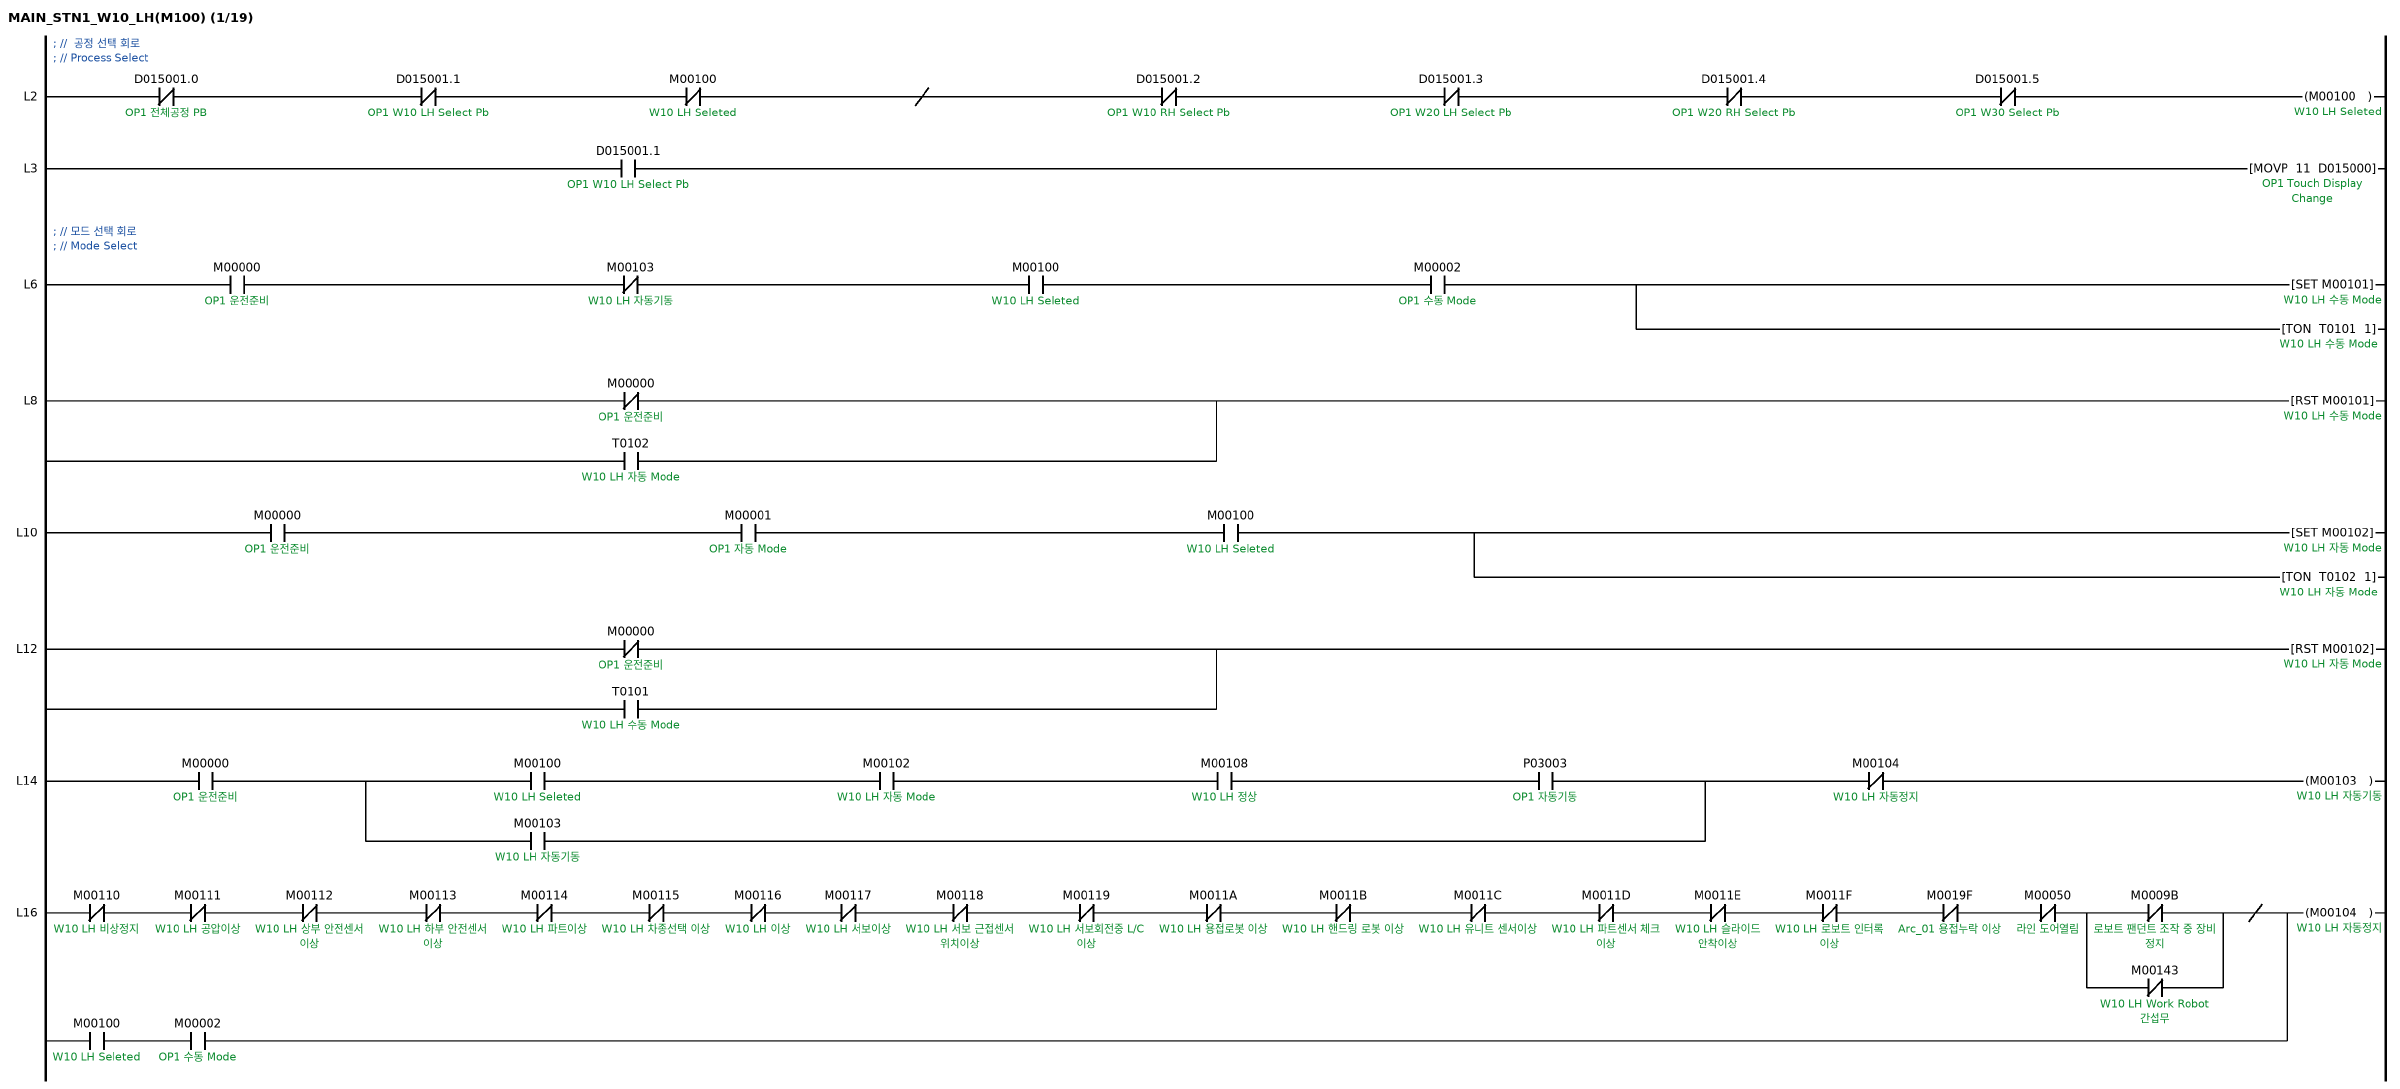
//   //  공정 선택 회로
//   // Process Select
; L2
LOAD NOT  D015001.0	// OP1 전체공정 PB
AND NOT   D015001.1	// OP1 W10 LH Select Pb
AND NOT   M00100	// W10 LH Seleted
NOT
AND NOT   D015001.2	// OP1 W10 RH Select Pb
AND NOT   D015001.3	// OP1 W20 LH Select Pb
AND NOT   D015001.4	// OP1 W20 RH Select Pb
AND NOT   D015001.5	// OP1 W30 Select Pb
OUT       M00100	// W10 LH Seleted
; L3
LOAD      D015001.1	// OP1 W10 LH Select Pb
MOVP      11 D015000	// OP1 Touch Display Change
// // 모드 선택 회로
//   // Mode Select
; L6
LOAD      M00000	// OP1 운전준비
AND NOT   M00103	// W10 LH 자동기동
AND       M00100	// W10 LH Seleted
AND       M00002	// OP1 수동 Mode
SET       M00101	// W10 LH 수동 Mode
TON       T0101 1	// W10 LH 수동 Mode
; L8
LOAD NOT  M00000	// OP1 운전준비
OR        T0102	// W10 LH 자동 Mode
RST       M00101	// W10 LH 수동 Mode
; L10
LOAD      M00000	// OP1 운전준비
AND       M00001	// OP1 자동 Mode
AND       M00100	// W10 LH Seleted
SET       M00102	// W10 LH 자동 Mode
TON       T0102 1	// W10 LH 자동 Mode
; L12
LOAD NOT  M00000	// OP1 운전준비
OR        T0101	// W10 LH 수동 Mode
RST       M00102	// W10 LH 자동 Mode
; L14
LOAD      M00000	// OP1 운전준비
LOAD      M00100	// W10 LH Seleted
AND       M00102	// W10 LH 자동 Mode
AND       M00108	// W10 LH 정상
AND       P03003	// OP1 자동기동
OR        M00103	// W10 LH 자동기동
AND LOAD
AND NOT   M00104	// W10 LH 자동정지
OUT       M00103	// W10 LH 자동기동
; L16
LOAD NOT  M00110	// W10 LH 비상정지
AND NOT   M00111	// W10 LH 공압이상
AND NOT   M00112	// W10 LH 상부 안전센서 이상
AND NOT   M00113	// W10 LH 하부 안전센서 이상
AND NOT   M00114	// W10 LH 파트이상
AND NOT   M00115	// W10 LH 차종선택 이상
AND NOT   M00116	// W10 LH 이상
AND NOT   M00117	// W10 LH 서보이상
AND NOT   M00118	// W10 LH 서보 근접센서 위치이상
AND NOT   M00119	// W10 LH 서보회전중 L/C 이상
AND NOT   M0011A	// W10 LH 용접로봇 이상
AND NOT   M0011B	// W10 LH 핸드링 로봇 이상
AND NOT   M0011C	// W10 LH 유니트 센서이상
AND NOT   M0011D	// W10 LH 파트센서 체크 이상
AND NOT   M0011E	// W10 LH 슬라이드 안착이상
AND NOT   M0011F	// W10 LH 로보트 인터록 이상
AND NOT   M0019F	// Arc_01 용접누락 이상
AND NOT   M00050	// 라인 도어열림
LOAD NOT  M0009B	// 로보트 팬던트 조작 중 장비 정지
OR NOT    M00143	// W10 LH Work Robot 간섭무
AND LOAD
NOT
LOAD      M00100	// W10 LH Seleted
AND       M00002	// OP1 수동 Mode
OR LOAD
OUT       M00104	// W10 LH 자동정지

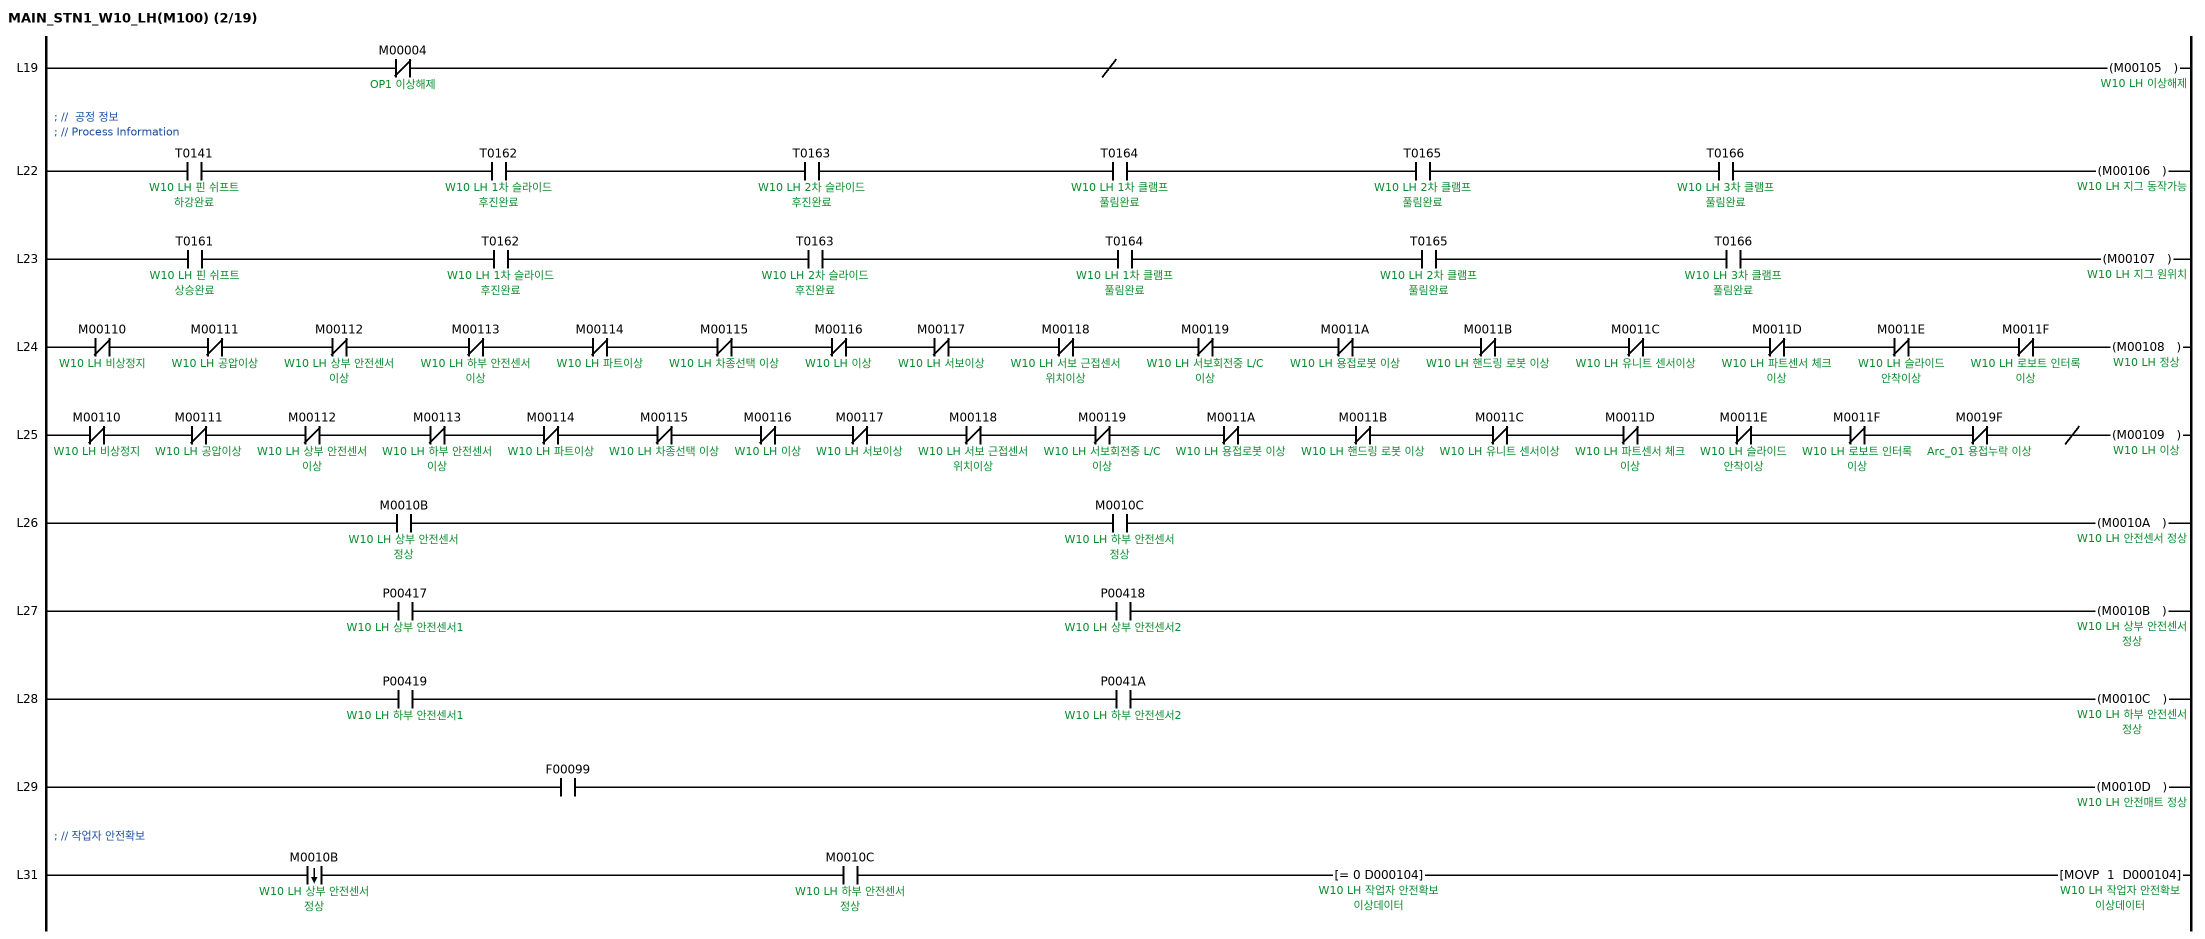
; L19
LOAD NOT  M00004	// OP1 이상해제
NOT
OUT       M00105	// W10 LH 이상해제
//   //  공정 정보
//   // Process Information
; L22
LOAD      T0141	// W10 LH 핀 쉬프트 하강완료
AND       T0162	// W10 LH 1차 슬라이드 후진완료
AND       T0163	// W10 LH 2차 슬라이드 후진완료
AND       T0164	// W10 LH 1차 클램프 풀림완료
AND       T0165	// W10 LH 2차 클램프 풀림완료
AND       T0166	// W10 LH 3차 클램프 풀림완료
OUT       M00106	// W10 LH 지그 동작가능
; L23
LOAD      T0161	// W10 LH 핀 쉬프트 상승완료
AND       T0162	// W10 LH 1차 슬라이드 후진완료
AND       T0163	// W10 LH 2차 슬라이드 후진완료
AND       T0164	// W10 LH 1차 클램프 풀림완료
AND       T0165	// W10 LH 2차 클램프 풀림완료
AND       T0166	// W10 LH 3차 클램프 풀림완료
OUT       M00107	// W10 LH 지그 원위치
; L24
LOAD NOT  M00110	// W10 LH 비상정지
AND NOT   M00111	// W10 LH 공압이상
AND NOT   M00112	// W10 LH 상부 안전센서 이상
AND NOT   M00113	// W10 LH 하부 안전센서 이상
AND NOT   M00114	// W10 LH 파트이상
AND NOT   M00115	// W10 LH 차종선택 이상
AND NOT   M00116	// W10 LH 이상
AND NOT   M00117	// W10 LH 서보이상
AND NOT   M00118	// W10 LH 서보 근접센서 위치이상
AND NOT   M00119	// W10 LH 서보회전중 L/C 이상
AND NOT   M0011A	// W10 LH 용접로봇 이상
AND NOT   M0011B	// W10 LH 핸드링 로봇 이상
AND NOT   M0011C	// W10 LH 유니트 센서이상
AND NOT   M0011D	// W10 LH 파트센서 체크 이상
AND NOT   M0011E	// W10 LH 슬라이드 안착이상
AND NOT   M0011F	// W10 LH 로보트 인터록 이상
OUT       M00108	// W10 LH 정상
; L25
LOAD NOT  M00110	// W10 LH 비상정지
AND NOT   M00111	// W10 LH 공압이상
AND NOT   M00112	// W10 LH 상부 안전센서 이상
AND NOT   M00113	// W10 LH 하부 안전센서 이상
AND NOT   M00114	// W10 LH 파트이상
AND NOT   M00115	// W10 LH 차종선택 이상
AND NOT   M00116	// W10 LH 이상
AND NOT   M00117	// W10 LH 서보이상
AND NOT   M00118	// W10 LH 서보 근접센서 위치이상
AND NOT   M00119	// W10 LH 서보회전중 L/C 이상
AND NOT   M0011A	// W10 LH 용접로봇 이상
AND NOT   M0011B	// W10 LH 핸드링 로봇 이상
AND NOT   M0011C	// W10 LH 유니트 센서이상
AND NOT   M0011D	// W10 LH 파트센서 체크 이상
AND NOT   M0011E	// W10 LH 슬라이드 안착이상
AND NOT   M0011F	// W10 LH 로보트 인터록 이상
AND NOT   M0019F	// Arc_01 용접누락 이상
NOT
OUT       M00109	// W10 LH 이상
; L26
LOAD      M0010B	// W10 LH 상부 안전센서 정상
AND       M0010C	// W10 LH 하부 안전센서 정상
OUT       M0010A	// W10 LH 안전센서 정상
; L27
LOAD      P00417	// W10 LH 상부 안전센서1
AND       P00418	// W10 LH 상부 안전센서2
OUT       M0010B	// W10 LH 상부 안전센서 정상
; L28
LOAD      P00419	// W10 LH 하부 안전센서1
AND       P0041A	// W10 LH 하부 안전센서2
OUT       M0010C	// W10 LH 하부 안전센서 정상
; L29
LOAD      F00099
OUT       M0010D	// W10 LH 안전매트 정상
//    // 작업자 안전확보
; L31
LOADN     M0010B	// W10 LH 상부 안전센서 정상
AND       M0010C	// W10 LH 하부 안전센서 정상
AND=      0 D000104	// W10 LH 작업자 안전확보 이상데이터
MOVP      1 D000104	// W10 LH 작업자 안전확보 이상데이터

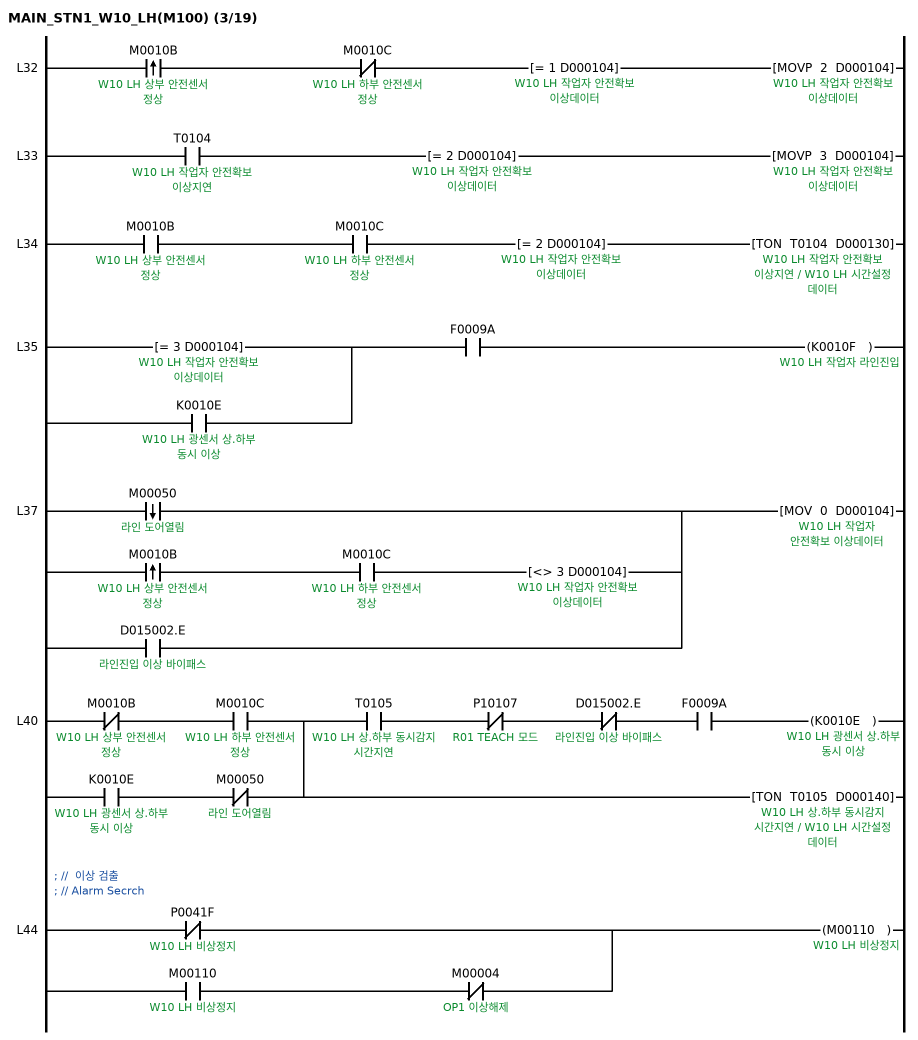
; L32
LOADP     M0010B	// W10 LH 상부 안전센서 정상
AND NOT   M0010C	// W10 LH 하부 안전센서 정상
AND=      1 D000104	// W10 LH 작업자 안전확보 이상데이터
MOVP      2 D000104	// W10 LH 작업자 안전확보 이상데이터
; L33
LOAD      T0104	// W10 LH 작업자 안전확보 이상지연
AND=      2 D000104	// W10 LH 작업자 안전확보 이상데이터
MOVP      3 D000104	// W10 LH 작업자 안전확보 이상데이터
; L34
LOAD      M0010B	// W10 LH 상부 안전센서 정상
AND       M0010C	// W10 LH 하부 안전센서 정상
AND=      2 D000104	// W10 LH 작업자 안전확보 이상데이터
TON       T0104 D000130	// W10 LH 작업자 안전확보 이상지연 / W10 LH 시간설정 데이터
; L35
LOAD=     3 D000104	// W10 LH 작업자 안전확보 이상데이터
OR        K0010E	// W10 LH 광센서 상.하부 동시 이상
AND       F0009A
OUT       K0010F	// W10 LH 작업자 라인진입
; L37
LOADN     M00050	// 라인 도어열림
LOADP     M0010B	// W10 LH 상부 안전센서 정상
AND       M0010C	// W10 LH 하부 안전센서 정상
AND<>     3 D000104	// W10 LH 작업자 안전확보 이상데이터
OR LOAD
OR        D015002.E	// 라인진입 이상 바이패스
MOV       0 D000104	// W10 LH 작업자 안전확보 이상데이터
; L40
LOAD NOT  M0010B	// W10 LH 상부 안전센서 정상
AND       M0010C	// W10 LH 하부 안전센서 정상
LOAD      K0010E	// W10 LH 광센서 상.하부 동시 이상
AND NOT   M00050	// 라인 도어열림
OR LOAD
MPUSH
AND       T0105	// W10 LH 상.하부 동시감지 시간지연
AND NOT   P10107	// R01 TEACH 모드
AND NOT   D015002.E	// 라인진입 이상 바이패스
AND       F0009A
OUT       K0010E	// W10 LH 광센서 상.하부 동시 이상
MPOP
TON       T0105 D000140	// W10 LH 상.하부 동시감지 시간지연 / W10 LH 시간설정 데이터
//   //  이상 검출
//   // Alarm Secrch
; L44
LOAD NOT  P0041F	// W10 LH 비상정지
LOAD      M00110	// W10 LH 비상정지
AND NOT   M00004	// OP1 이상해제
OR LOAD
OUT       M00110	// W10 LH 비상정지

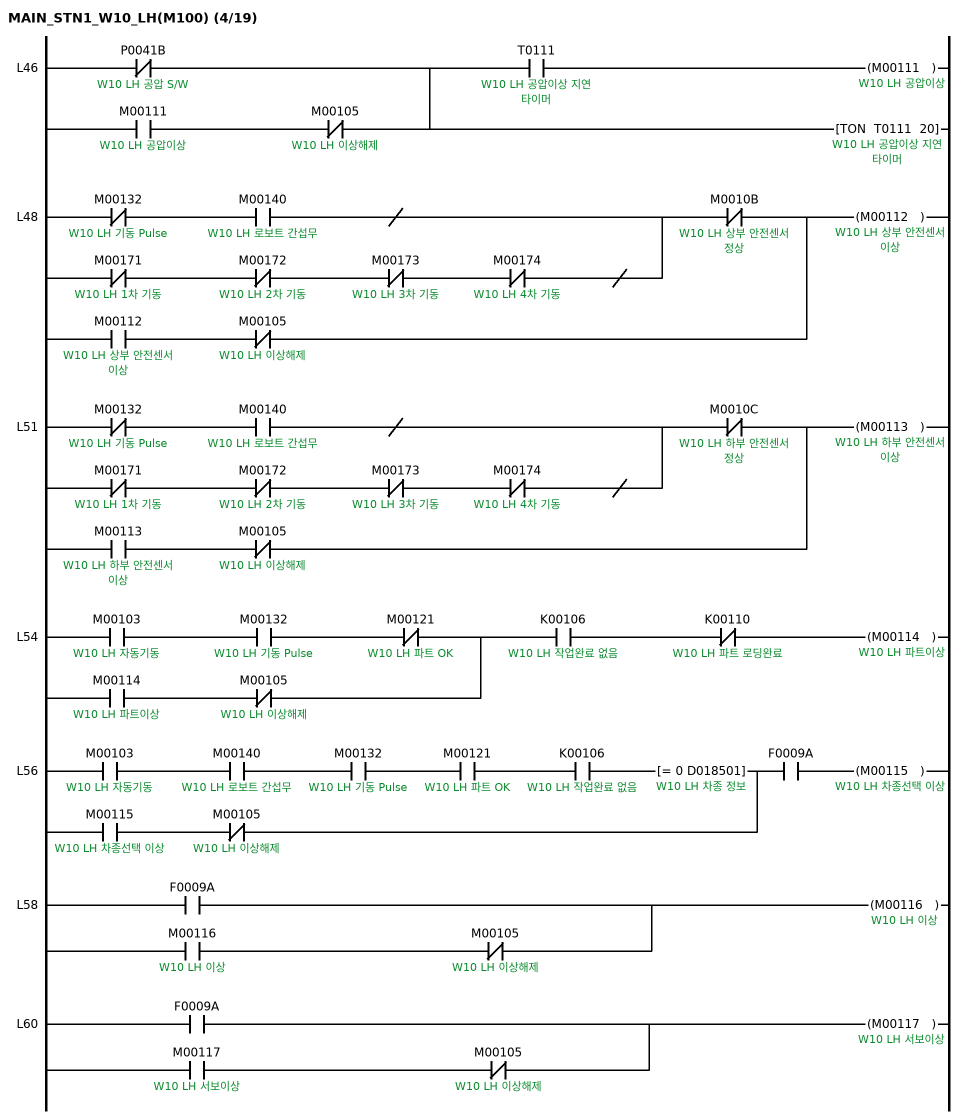
; L46
LOAD NOT  P0041B	// W10 LH 공압 S/W
LOAD      M00111	// W10 LH 공압이상
AND NOT   M00105	// W10 LH 이상해제
OR LOAD
MPUSH
AND       T0111	// W10 LH 공압이상 지연 타이머
OUT       M00111	// W10 LH 공압이상
MPOP
TON       T0111 20	// W10 LH 공압이상 지연 타이머
; L48
LOAD NOT  M00132	// W10 LH 기동 Pulse
AND       M00140	// W10 LH 로보트 간섭무
NOT
LOAD NOT  M00171	// W10 LH 1차 기동
AND NOT   M00172	// W10 LH 2차 기동
AND NOT   M00173	// W10 LH 3차 기동
AND NOT   M00174	// W10 LH 4차 기동
NOT
OR LOAD
AND NOT   M0010B	// W10 LH 상부 안전센서 정상
LOAD      M00112	// W10 LH 상부 안전센서 이상
AND NOT   M00105	// W10 LH 이상해제
OR LOAD
OUT       M00112	// W10 LH 상부 안전센서 이상
; L51
LOAD NOT  M00132	// W10 LH 기동 Pulse
AND       M00140	// W10 LH 로보트 간섭무
NOT
LOAD NOT  M00171	// W10 LH 1차 기동
AND NOT   M00172	// W10 LH 2차 기동
AND NOT   M00173	// W10 LH 3차 기동
AND NOT   M00174	// W10 LH 4차 기동
NOT
OR LOAD
AND NOT   M0010C	// W10 LH 하부 안전센서 정상
LOAD      M00113	// W10 LH 하부 안전센서 이상
AND NOT   M00105	// W10 LH 이상해제
OR LOAD
OUT       M00113	// W10 LH 하부 안전센서 이상
; L54
LOAD      M00103	// W10 LH 자동기동
AND       M00132	// W10 LH 기동 Pulse
AND NOT   M00121	// W10 LH 파트 OK
LOAD      M00114	// W10 LH 파트이상
AND NOT   M00105	// W10 LH 이상해제
OR LOAD
AND       K00106	// W10 LH 작업완료 없음
AND NOT   K00110	// W10 LH 파트 로딩완료
OUT       M00114	// W10 LH 파트이상
; L56
LOAD      M00103	// W10 LH 자동기동
AND       M00140	// W10 LH 로보트 간섭무
AND       M00132	// W10 LH 기동 Pulse
AND       M00121	// W10 LH 파트 OK
AND       K00106	// W10 LH 작업완료 없음
AND=      0 D018501	// W10 LH 차종 정보
LOAD      M00115	// W10 LH 차종선택 이상
AND NOT   M00105	// W10 LH 이상해제
OR LOAD
AND       F0009A
OUT       M00115	// W10 LH 차종선택 이상
; L58
LOAD      F0009A
LOAD      M00116	// W10 LH 이상
AND NOT   M00105	// W10 LH 이상해제
OR LOAD
OUT       M00116	// W10 LH 이상
; L60
LOAD      F0009A
LOAD      M00117	// W10 LH 서보이상
AND NOT   M00105	// W10 LH 이상해제
OR LOAD
OUT       M00117	// W10 LH 서보이상

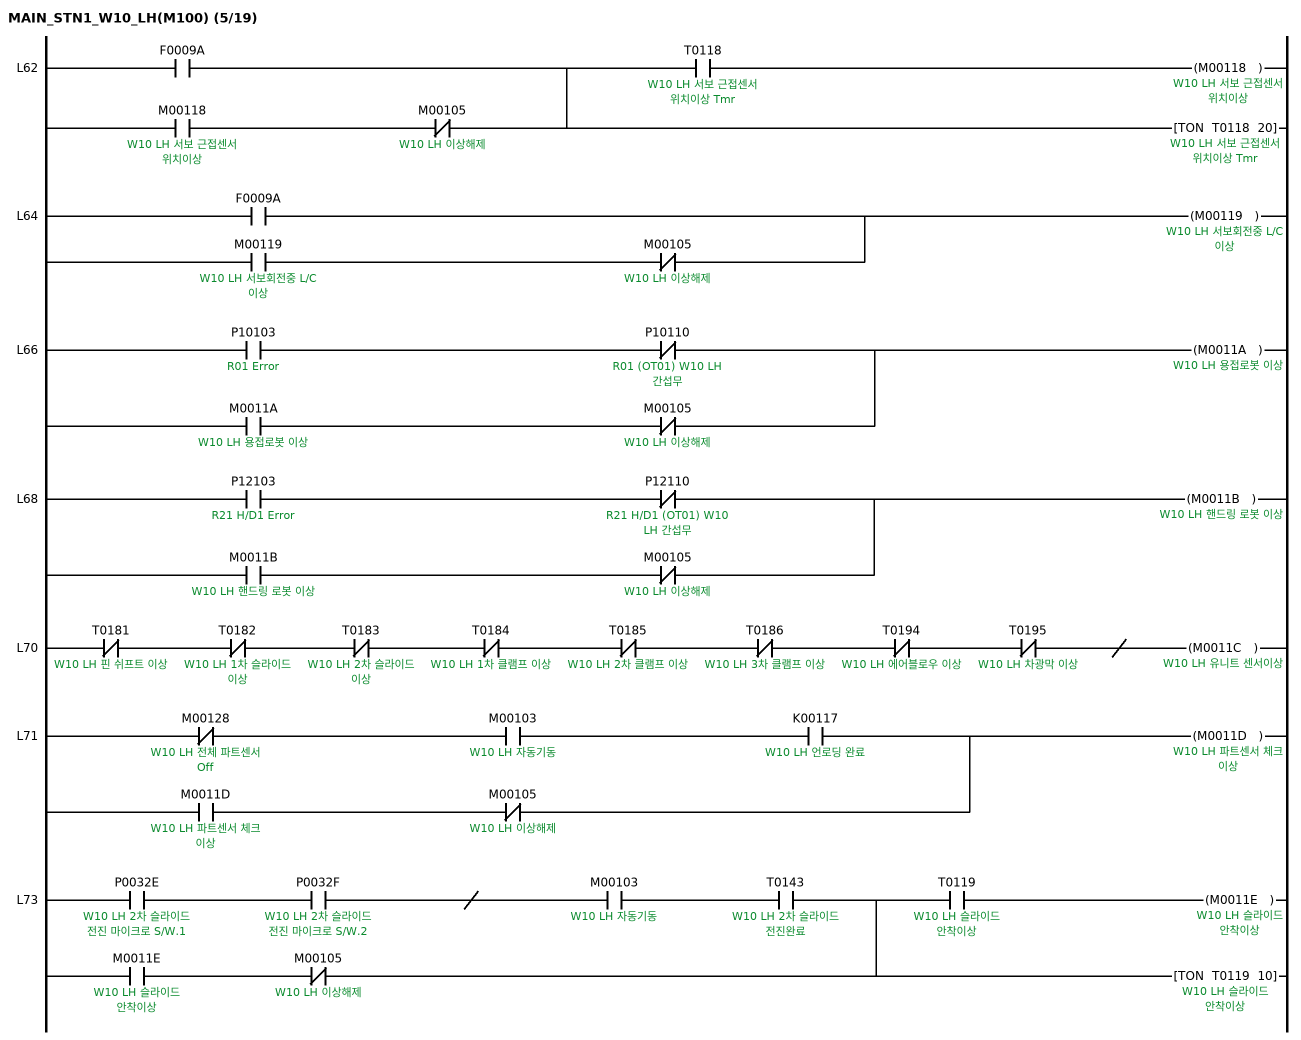
; L62
LOAD      F0009A
LOAD      M00118	// W10 LH 서보 근접센서 위치이상
AND NOT   M00105	// W10 LH 이상해제
OR LOAD
MPUSH
AND       T0118	// W10 LH 서보 근접센서 위치이상 Tmr
OUT       M00118	// W10 LH 서보 근접센서 위치이상
MPOP
TON       T0118 20	// W10 LH 서보 근접센서 위치이상 Tmr
; L64
LOAD      F0009A
LOAD      M00119	// W10 LH 서보회전중 L/C 이상
AND NOT   M00105	// W10 LH 이상해제
OR LOAD
OUT       M00119	// W10 LH 서보회전중 L/C 이상
; L66
LOAD      P10103	// R01 Error
AND NOT   P10110	// R01 (OT01) W10 LH 간섭무
LOAD      M0011A	// W10 LH 용접로봇 이상
AND NOT   M00105	// W10 LH 이상해제
OR LOAD
OUT       M0011A	// W10 LH 용접로봇 이상
; L68
LOAD      P12103	// R21 H/D1 Error
AND NOT   P12110	// R21 H/D1 (OT01) W10 LH 간섭무
LOAD      M0011B	// W10 LH 핸드링 로봇 이상
AND NOT   M00105	// W10 LH 이상해제
OR LOAD
OUT       M0011B	// W10 LH 핸드링 로봇 이상
; L70
LOAD NOT  T0181	// W10 LH 핀 쉬프트 이상
AND NOT   T0182	// W10 LH 1차 슬라이드 이상
AND NOT   T0183	// W10 LH 2차 슬라이드 이상
AND NOT   T0184	// W10 LH 1차 클램프 이상
AND NOT   T0185	// W10 LH 2차 클램프 이상
AND NOT   T0186	// W10 LH 3차 클램프 이상
AND NOT   T0194	// W10 LH 에어블로우 이상
AND NOT   T0195	// W10 LH 차광막 이상
NOT
OUT       M0011C	// W10 LH 유니트 센서이상
; L71
LOAD NOT  M00128	// W10 LH 전체 파트센서 Off
AND       M00103	// W10 LH 자동기동
AND       K00117	// W10 LH 언로딩 완료
LOAD      M0011D	// W10 LH 파트센서 체크 이상
AND NOT   M00105	// W10 LH 이상해제
OR LOAD
OUT       M0011D	// W10 LH 파트센서 체크 이상
; L73
LOAD      P0032E	// W10 LH 2차 슬라이드 전진 마이크로 S/W.1
AND       P0032F	// W10 LH 2차 슬라이드 전진 마이크로 S/W.2
NOT
AND       M00103	// W10 LH 자동기동
AND       T0143	// W10 LH 2차 슬라이드 전진완료
LOAD      M0011E	// W10 LH 슬라이드 안착이상
AND NOT   M00105	// W10 LH 이상해제
OR LOAD
MPUSH
AND       T0119	// W10 LH 슬라이드 안착이상
OUT       M0011E	// W10 LH 슬라이드 안착이상
MPOP
TON       T0119 10	// W10 LH 슬라이드 안착이상

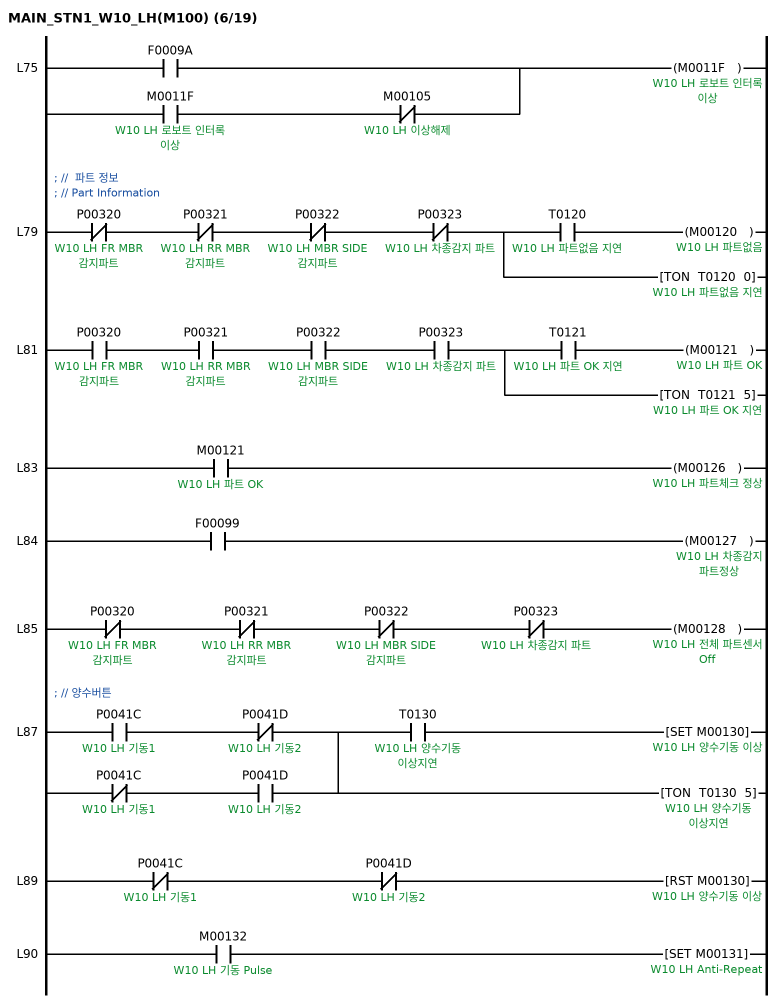
; L75
LOAD      F0009A
LOAD      M0011F	// W10 LH 로보트 인터록 이상
AND NOT   M00105	// W10 LH 이상해제
OR LOAD
OUT       M0011F	// W10 LH 로보트 인터록 이상
//   //  파트 정보
//   // Part Information
; L79
LOAD NOT  P00320	// W10 LH FR MBR 감지파트
AND NOT   P00321	// W10 LH RR MBR 감지파트
AND NOT   P00322	// W10 LH MBR SIDE 감지파트
AND NOT   P00323	// W10 LH 차종감지 파트
MPUSH
AND       T0120	// W10 LH 파트없음 지연
OUT       M00120	// W10 LH 파트없음
MPOP
TON       T0120 0	// W10 LH 파트없음 지연
; L81
LOAD      P00320	// W10 LH FR MBR 감지파트
AND       P00321	// W10 LH RR MBR 감지파트
AND       P00322	// W10 LH MBR SIDE 감지파트
AND       P00323	// W10 LH 차종감지 파트
MPUSH
AND       T0121	// W10 LH 파트 OK 지연
OUT       M00121	// W10 LH 파트 OK
MPOP
TON       T0121 5	// W10 LH 파트 OK 지연
; L83
LOAD      M00121	// W10 LH 파트 OK
OUT       M00126	// W10 LH 파트체크 정상
; L84
LOAD      F00099
OUT       M00127	// W10 LH 차종감지 파트정상
; L85
LOAD NOT  P00320	// W10 LH FR MBR 감지파트
AND NOT   P00321	// W10 LH RR MBR 감지파트
AND NOT   P00322	// W10 LH MBR SIDE 감지파트
AND NOT   P00323	// W10 LH 차종감지 파트
OUT       M00128	// W10 LH 전체 파트센서 Off
//   // 양수버튼
; L87
LOAD      P0041C	// W10 LH 기동1
AND NOT   P0041D	// W10 LH 기동2
LOAD NOT  P0041C	// W10 LH 기동1
AND       P0041D	// W10 LH 기동2
OR LOAD
MPUSH
AND       T0130	// W10 LH 양수기동 이상지연
SET       M00130	// W10 LH 양수기동 이상
MPOP
TON       T0130 5	// W10 LH 양수기동 이상지연
; L89
LOAD NOT  P0041C	// W10 LH 기동1
AND NOT   P0041D	// W10 LH 기동2
RST       M00130	// W10 LH 양수기동 이상
; L90
LOAD      M00132	// W10 LH 기동 Pulse
SET       M00131	// W10 LH Anti-Repeat

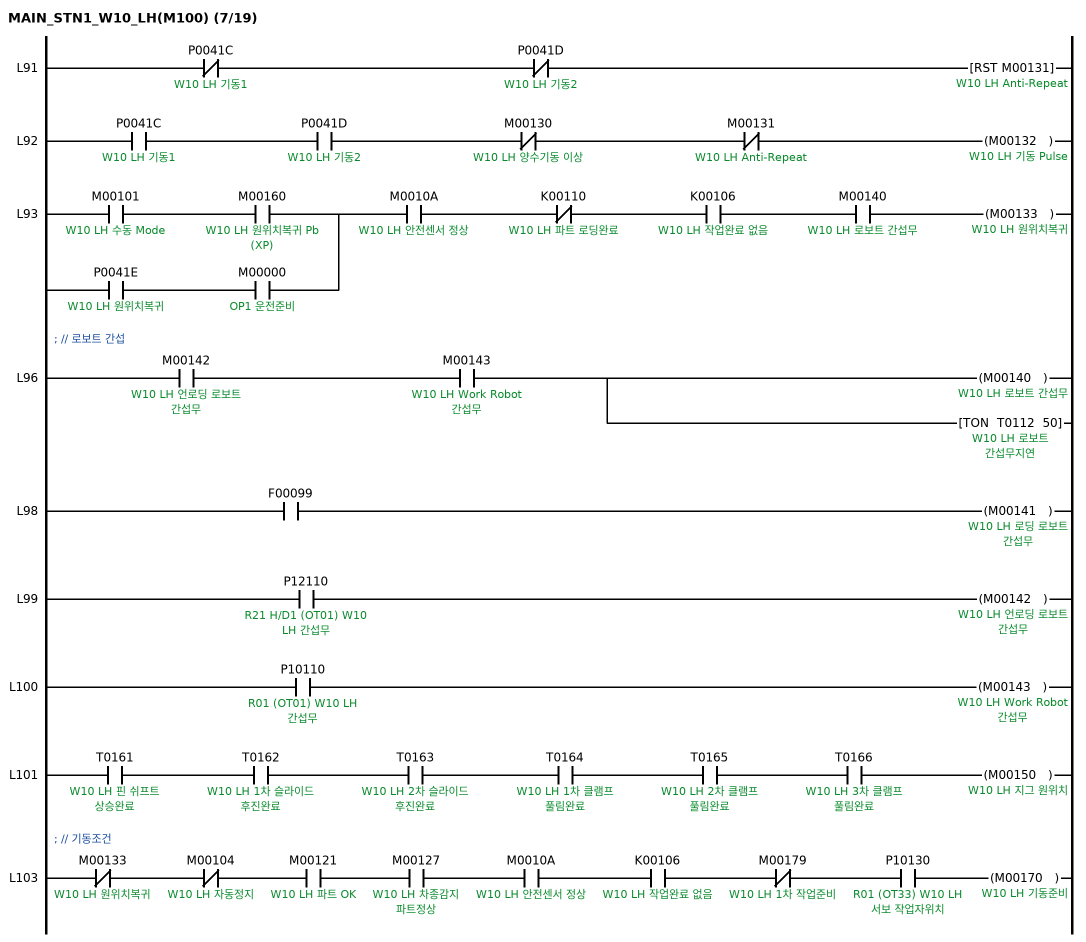
; L91
LOAD NOT  P0041C	// W10 LH 기동1
AND NOT   P0041D	// W10 LH 기동2
RST       M00131	// W10 LH Anti-Repeat
; L92
LOAD      P0041C	// W10 LH 기동1
AND       P0041D	// W10 LH 기동2
AND NOT   M00130	// W10 LH 양수기동 이상
AND NOT   M00131	// W10 LH Anti-Repeat
OUT       M00132	// W10 LH 기동 Pulse
; L93
LOAD      M00101	// W10 LH 수동 Mode
AND       M00160	// W10 LH 원위치복귀 Pb (XP)
LOAD      P0041E	// W10 LH 원위치복귀
AND       M00000	// OP1 운전준비
OR LOAD
AND       M0010A	// W10 LH 안전센서 정상
AND NOT   K00110	// W10 LH 파트 로딩완료
AND       K00106	// W10 LH 작업완료 없음
AND       M00140	// W10 LH 로보트 간섭무
OUT       M00133	// W10 LH 원위치복귀
//   // 로보트 간섭
; L96
LOAD      M00142	// W10 LH 언로딩 로보트 간섭무
AND       M00143	// W10 LH Work Robot 간섭무
OUT       M00140	// W10 LH 로보트 간섭무
TON       T0112 50	// W10 LH 로보트 간섭무지연
; L98
LOAD      F00099
OUT       M00141	// W10 LH 로딩 로보트 간섭무
; L99
LOAD      P12110	// R21 H/D1 (OT01) W10 LH 간섭무
OUT       M00142	// W10 LH 언로딩 로보트 간섭무
; L100
LOAD      P10110	// R01 (OT01) W10 LH 간섭무
OUT       M00143	// W10 LH Work Robot 간섭무
; L101
LOAD      T0161	// W10 LH 핀 쉬프트 상승완료
AND       T0162	// W10 LH 1차 슬라이드 후진완료
AND       T0163	// W10 LH 2차 슬라이드 후진완료
AND       T0164	// W10 LH 1차 클램프 풀림완료
AND       T0165	// W10 LH 2차 클램프 풀림완료
AND       T0166	// W10 LH 3차 클램프 풀림완료
OUT       M00150	// W10 LH 지그 원위치
//   // 기동조건
; L103
LOAD NOT  M00133	// W10 LH 원위치복귀
AND NOT   M00104	// W10 LH 자동정지
AND       M00121	// W10 LH 파트 OK
AND       M00127	// W10 LH 차종감지 파트정상
AND       M0010A	// W10 LH 안전센서 정상
AND       K00106	// W10 LH 작업완료 없음
AND NOT   M00179	// W10 LH 1차 작업준비
AND       P10130	// R01 (OT33) W10 LH 서보 작업자위치
OUT       M00170	// W10 LH 기동준비

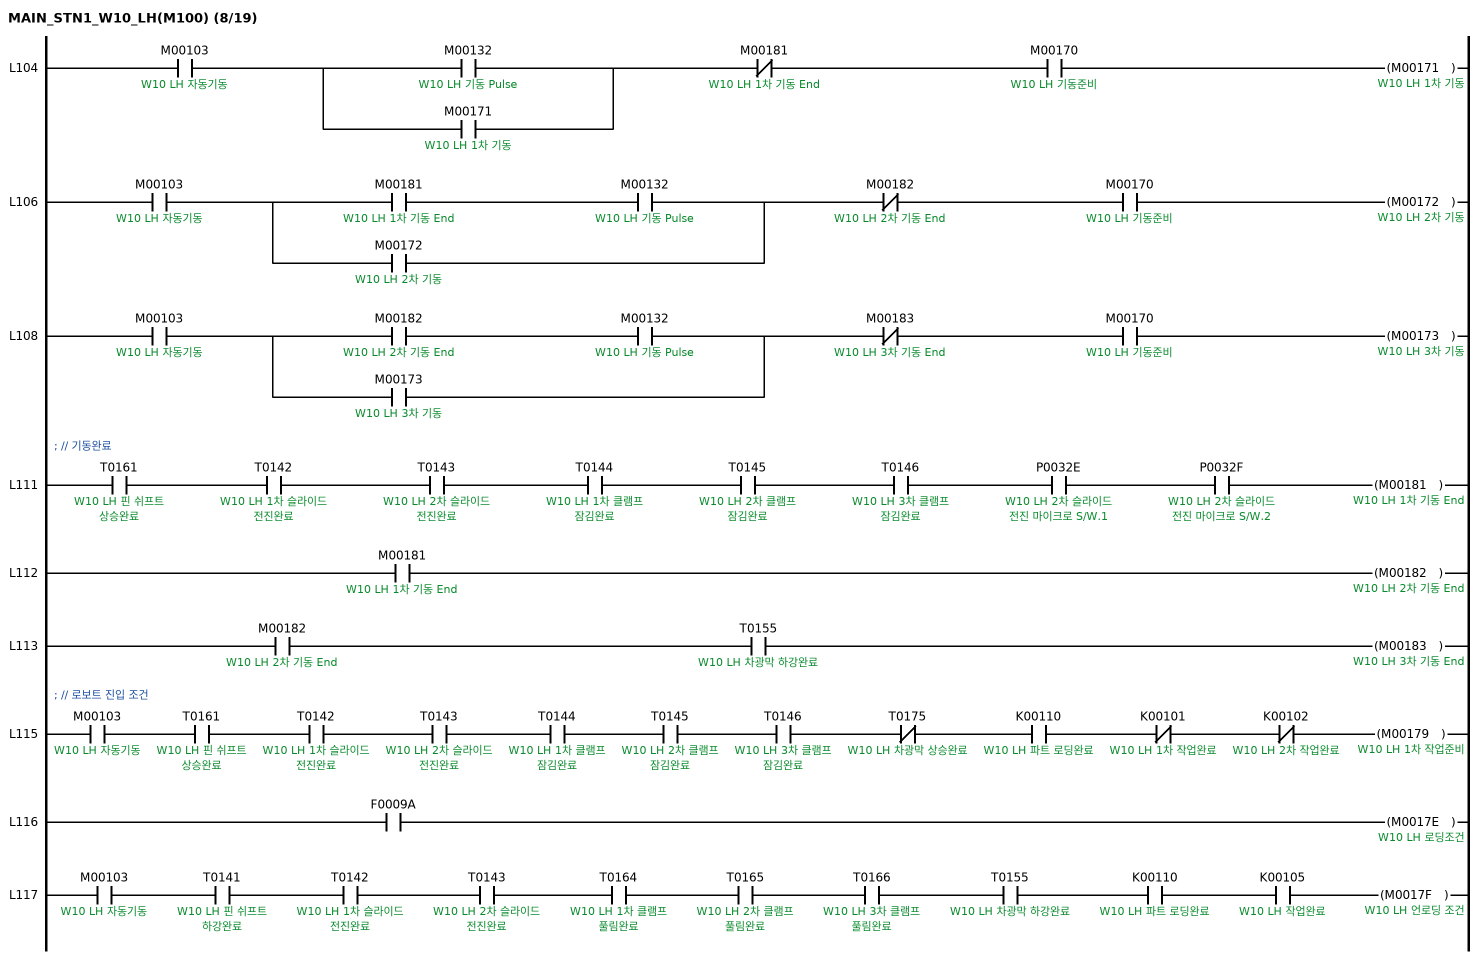
; L104
LOAD      M00103	// W10 LH 자동기동
LOAD      M00132	// W10 LH 기동 Pulse
OR        M00171	// W10 LH 1차 기동
AND LOAD
AND NOT   M00181	// W10 LH 1차 기동 End
AND       M00170	// W10 LH 기동준비
OUT       M00171	// W10 LH 1차 기동
; L106
LOAD      M00103	// W10 LH 자동기동
LOAD      M00181	// W10 LH 1차 기동 End
AND       M00132	// W10 LH 기동 Pulse
OR        M00172	// W10 LH 2차 기동
AND LOAD
AND NOT   M00182	// W10 LH 2차 기동 End
AND       M00170	// W10 LH 기동준비
OUT       M00172	// W10 LH 2차 기동
; L108
LOAD      M00103	// W10 LH 자동기동
LOAD      M00182	// W10 LH 2차 기동 End
AND       M00132	// W10 LH 기동 Pulse
OR        M00173	// W10 LH 3차 기동
AND LOAD
AND NOT   M00183	// W10 LH 3차 기동 End
AND       M00170	// W10 LH 기동준비
OUT       M00173	// W10 LH 3차 기동
//   // 기동완료
; L111
LOAD      T0161	// W10 LH 핀 쉬프트 상승완료
AND       T0142	// W10 LH 1차 슬라이드 전진완료
AND       T0143	// W10 LH 2차 슬라이드 전진완료
AND       T0144	// W10 LH 1차 클램프 잠김완료
AND       T0145	// W10 LH 2차 클램프 잠김완료
AND       T0146	// W10 LH 3차 클램프 잠김완료
AND       P0032E	// W10 LH 2차 슬라이드 전진 마이크로 S/W.1
AND       P0032F	// W10 LH 2차 슬라이드 전진 마이크로 S/W.2
OUT       M00181	// W10 LH 1차 기동 End
; L112
LOAD      M00181	// W10 LH 1차 기동 End
OUT       M00182	// W10 LH 2차 기동 End
; L113
LOAD      M00182	// W10 LH 2차 기동 End
AND       T0155	// W10 LH 차광막 하강완료
OUT       M00183	// W10 LH 3차 기동 End
//   // 로보트 진입 조건
; L115
LOAD      M00103	// W10 LH 자동기동
AND       T0161	// W10 LH 핀 쉬프트 상승완료
AND       T0142	// W10 LH 1차 슬라이드 전진완료
AND       T0143	// W10 LH 2차 슬라이드 전진완료
AND       T0144	// W10 LH 1차 클램프 잠김완료
AND       T0145	// W10 LH 2차 클램프 잠김완료
AND       T0146	// W10 LH 3차 클램프 잠김완료
AND NOT   T0175	// W10 LH 차광막 상승완료
AND       K00110	// W10 LH 파트 로딩완료
AND NOT   K00101	// W10 LH 1차 작업완료
AND NOT   K00102	// W10 LH 2차 작업완료
OUT       M00179	// W10 LH 1차 작업준비
; L116
LOAD      F0009A
OUT       M0017E	// W10 LH 로딩조건
; L117
LOAD      M00103	// W10 LH 자동기동
AND       T0141	// W10 LH 핀 쉬프트 하강완료
AND       T0142	// W10 LH 1차 슬라이드 전진완료
AND       T0143	// W10 LH 2차 슬라이드 전진완료
AND       T0164	// W10 LH 1차 클램프 풀림완료
AND       T0165	// W10 LH 2차 클램프 풀림완료
AND       T0166	// W10 LH 3차 클램프 풀림완료
AND       T0155	// W10 LH 차광막 하강완료
AND       K00110	// W10 LH 파트 로딩완료
AND       K00105	// W10 LH 작업완료
OUT       M0017F	// W10 LH 언로딩 조건

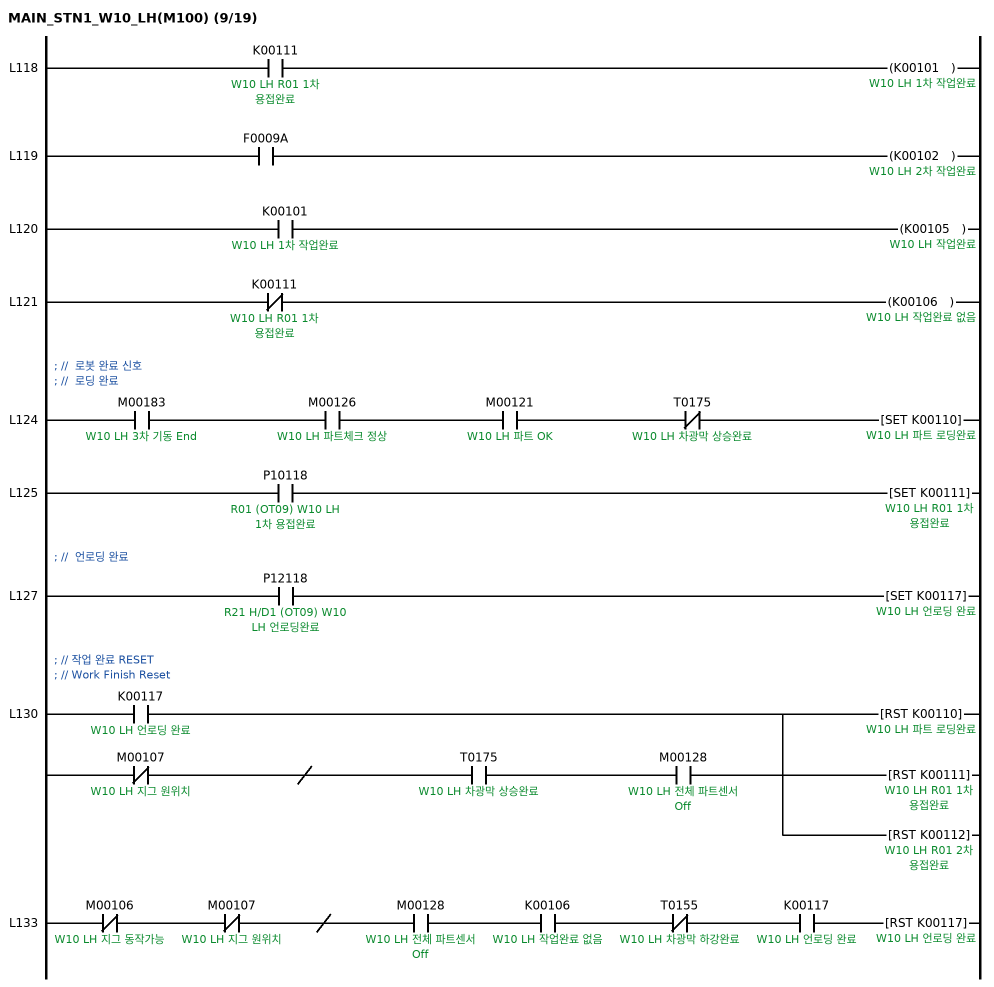
; L118
LOAD      K00111	// W10 LH R01 1차 용접완료
OUT       K00101	// W10 LH 1차 작업완료
; L119
LOAD      F0009A
OUT       K00102	// W10 LH 2차 작업완료
; L120
LOAD      K00101	// W10 LH 1차 작업완료
OUT       K00105	// W10 LH 작업완료
; L121
LOAD NOT  K00111	// W10 LH R01 1차 용접완료
OUT       K00106	// W10 LH 작업완료 없음
//   //  로봇 완료 신호
//   //  로딩 완료
; L124
LOAD      M00183	// W10 LH 3차 기동 End
AND       M00126	// W10 LH 파트체크 정상
AND       M00121	// W10 LH 파트 OK
AND NOT   T0175	// W10 LH 차광막 상승완료
SET       K00110	// W10 LH 파트 로딩완료
; L125
LOAD      P10118	// R01 (OT09) W10 LH 1차 용접완료
SET       K00111	// W10 LH R01 1차 용접완료
//   //  언로딩 완료
; L127
LOAD      P12118	// R21 H/D1 (OT09) W10 LH 언로딩완료
SET       K00117	// W10 LH 언로딩 완료
//     // 작업 완료 RESET
//   // Work Finish Reset
; L130
LOAD      K00117	// W10 LH 언로딩 완료
LOAD NOT  M00107	// W10 LH 지그 원위치
NOT
AND       T0175	// W10 LH 차광막 상승완료
AND       M00128	// W10 LH 전체 파트센서 Off
OR LOAD
RST       K00110	// W10 LH 파트 로딩완료
RST       K00111	// W10 LH R01 1차 용접완료
RST       K00112	// W10 LH R01 2차 용접완료
; L133
LOAD NOT  M00106	// W10 LH 지그 동작가능
AND NOT   M00107	// W10 LH 지그 원위치
NOT
AND       M00128	// W10 LH 전체 파트센서 Off
AND       K00106	// W10 LH 작업완료 없음
AND NOT   T0155	// W10 LH 차광막 하강완료
AND       K00117	// W10 LH 언로딩 완료
RST       K00117	// W10 LH 언로딩 완료

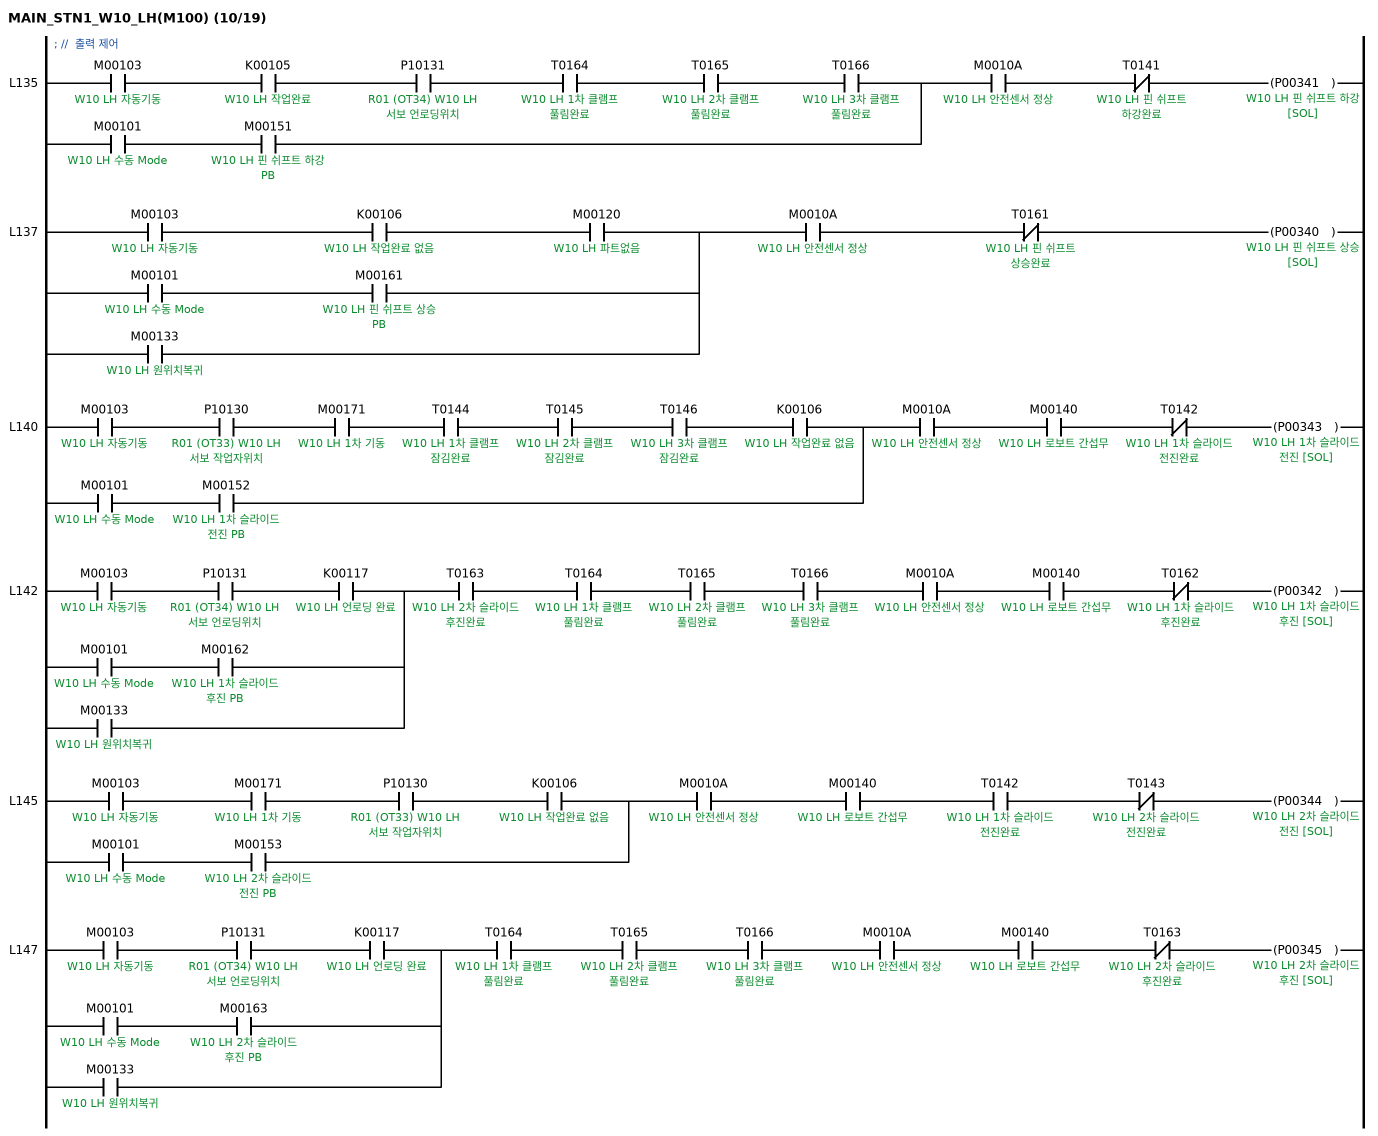
//     //  출력 제어
; L135
LOAD      M00103	// W10 LH 자동기동
AND       K00105	// W10 LH 작업완료
AND       P10131	// R01 (OT34) W10 LH 서보 언로딩위치
AND       T0164	// W10 LH 1차 클램프 풀림완료
AND       T0165	// W10 LH 2차 클램프 풀림완료
AND       T0166	// W10 LH 3차 클램프 풀림완료
LOAD      M00101	// W10 LH 수동 Mode
AND       M00151	// W10 LH 핀 쉬프트 하강 PB
OR LOAD
AND       M0010A	// W10 LH 안전센서 정상
AND NOT   T0141	// W10 LH 핀 쉬프트 하강완료
OUT       P00341	// W10 LH 핀 쉬프트 하강 [SOL]
; L137
LOAD      M00103	// W10 LH 자동기동
AND       K00106	// W10 LH 작업완료 없음
AND       M00120	// W10 LH 파트없음
LOAD      M00101	// W10 LH 수동 Mode
AND       M00161	// W10 LH 핀 쉬프트 상승 PB
OR LOAD
OR        M00133	// W10 LH 원위치복귀
AND       M0010A	// W10 LH 안전센서 정상
AND NOT   T0161	// W10 LH 핀 쉬프트 상승완료
OUT       P00340	// W10 LH 핀 쉬프트 상승 [SOL]
; L140
LOAD      M00103	// W10 LH 자동기동
AND       P10130	// R01 (OT33) W10 LH 서보 작업자위치
AND       M00171	// W10 LH 1차 기동
AND       T0144	// W10 LH 1차 클램프 잠김완료
AND       T0145	// W10 LH 2차 클램프 잠김완료
AND       T0146	// W10 LH 3차 클램프 잠김완료
AND       K00106	// W10 LH 작업완료 없음
LOAD      M00101	// W10 LH 수동 Mode
AND       M00152	// W10 LH 1차 슬라이드 전진 PB
OR LOAD
AND       M0010A	// W10 LH 안전센서 정상
AND       M00140	// W10 LH 로보트 간섭무
AND NOT   T0142	// W10 LH 1차 슬라이드 전진완료
OUT       P00343	// W10 LH 1차 슬라이드 전진 [SOL]
; L142
LOAD      M00103	// W10 LH 자동기동
AND       P10131	// R01 (OT34) W10 LH 서보 언로딩위치
AND       K00117	// W10 LH 언로딩 완료
LOAD      M00101	// W10 LH 수동 Mode
AND       M00162	// W10 LH 1차 슬라이드 후진 PB
OR LOAD
OR        M00133	// W10 LH 원위치복귀
AND       T0163	// W10 LH 2차 슬라이드 후진완료
AND       T0164	// W10 LH 1차 클램프 풀림완료
AND       T0165	// W10 LH 2차 클램프 풀림완료
AND       T0166	// W10 LH 3차 클램프 풀림완료
AND       M0010A	// W10 LH 안전센서 정상
AND       M00140	// W10 LH 로보트 간섭무
AND NOT   T0162	// W10 LH 1차 슬라이드 후진완료
OUT       P00342	// W10 LH 1차 슬라이드 후진 [SOL]
; L145
LOAD      M00103	// W10 LH 자동기동
AND       M00171	// W10 LH 1차 기동
AND       P10130	// R01 (OT33) W10 LH 서보 작업자위치
AND       K00106	// W10 LH 작업완료 없음
LOAD      M00101	// W10 LH 수동 Mode
AND       M00153	// W10 LH 2차 슬라이드 전진 PB
OR LOAD
AND       M0010A	// W10 LH 안전센서 정상
AND       M00140	// W10 LH 로보트 간섭무
AND       T0142	// W10 LH 1차 슬라이드 전진완료
AND NOT   T0143	// W10 LH 2차 슬라이드 전진완료
OUT       P00344	// W10 LH 2차 슬라이드 전진 [SOL]
; L147
LOAD      M00103	// W10 LH 자동기동
AND       P10131	// R01 (OT34) W10 LH 서보 언로딩위치
AND       K00117	// W10 LH 언로딩 완료
LOAD      M00101	// W10 LH 수동 Mode
AND       M00163	// W10 LH 2차 슬라이드 후진 PB
OR LOAD
OR        M00133	// W10 LH 원위치복귀
AND       T0164	// W10 LH 1차 클램프 풀림완료
AND       T0165	// W10 LH 2차 클램프 풀림완료
AND       T0166	// W10 LH 3차 클램프 풀림완료
AND       M0010A	// W10 LH 안전센서 정상
AND       M00140	// W10 LH 로보트 간섭무
AND NOT   T0163	// W10 LH 2차 슬라이드 후진완료
OUT       P00345	// W10 LH 2차 슬라이드 후진 [SOL]

